	                    #sFB_Conveyor730(iUDT_ConveyorConfiguration := #iUDT_Configuration."730".Conveyor,
	                                     idi_PECEoSDistance := #iUDT_Configuration."730".PEC_Eos.Distance,
	                                     idi_PECBoSDistance := 0,
	                                     ii_ExternalSpeed := 0,
	                                     ix_SafetyOk := #ix_SafetyOk,
	                                     ix_24vOk := #ix_24vOk,
	                                     ix_400vOk := #ix_400vOk,
	                                     ix_HardwareOk := #ix_HardwareOk,
	                                     ix_PECEoS := #iqUDT_WorkstationStatus."730".PEC_EoS.PEC,
	                                     ix_PECBoS := TRUE,
	                                     ix_ReverseDirection := FALSE,
	                                     ix_ExternalRequestDieBack := FALSE,
	                                     ix_ExternalRequestHold := #sx_RightExternalRequestHold730,
	                                     ix_ResetEnergySave := FALSE,
	                                     qUDT_HMIStatus => #iqUDT_WorkstationStatus."730".Conveyor,
	                                     qUDT_Status => #iqUDT_WorkstationCommonStatus."730",
	                                     iqUDT_EquipmentControl := #iqUDT_EquipmentControl,
	                                     iqUDT_ConveyorCommand := #iqUDT_WorkstationCommands."730".Conveyor,
	                                     iqUDT_ConveyorInterface := #sUDT_Interface730,
	                                     iqUDT_HandShakeUp := #sUDT_Handshake720,
	                                     iqUDT_HandShake := #sUDT_Handshake730,
	                                     iqUDT_Statistics := #iqUDT_WorkstationStatistics."730".Conveyor);
	                END_REGION

	                REGION MCO

	                    #sFB_MCOConveyLinxAixController730(iUDT_AixConfig := #iUDT_Configuration."730".MCO_M01,
	                                                       iUDT_AixInputsModule := #iUDT_MotorInput730,
	                                                       ix_24vOk := #ix_24vOk,
	                                                       ix_SimulationModeActive := "DB_Memory".Simulation,
	                                                       ii_MotorPositionId := 1,
	                                                       qUDT_HMIStatus => #iqUDT_WorkstationStatus."730".MCO_M01,
	                                                       iqUDT_AixOutputsModule := #iqUDT_MotorOutput730,
	                                                       iqUDT_ConveyorInterface := #sUDT_Interface730,
	                                                       iqUDT_MCOStatistics := #iqUDT_WorkstationStatistics."730".MCO_M01);
	                END_REGION
	            END_REGION

	            REGION 740

	                REGION Displacement

	                    #sFB_Displacement740(#sUDT_Interface740);

	                END_REGION

	                REGION EOS
	                    #sFB_PEC740(ix_PEC := NOT #iUDT_MotorInput730.AllSensorPortInputs.RightSensor,
	                                iUDT_PECConfiguration := #iUDT_Configuration."740".PEC_Eos,
	                                qx_PECFiltered => #tx_dummy,
	                                qUDT_HMIStatus => #iqUDT_WorkstationStatus."740".PEC_EoS,
	                                iqUDT_ConveyorInterface := #sUDT_Interface740,
	                                iqUDT_PECStatistics := #iqUDT_WorkstationStatistics."740".PEC_EoS);


	                END_REGION


	                REGION Conveyor

	                    #sFB_Conveyor740(iUDT_ConveyorConfiguration := #iUDT_Configuration."740".Conveyor,
	                                     idi_PECEoSDistance := #iUDT_Configuration."740".PEC_Eos.Distance,
	                                     idi_PECBoSDistance := 0,
	                                     ii_ExternalSpeed := 0,
	                                     ix_SafetyOk := #ix_SafetyOk,
	                                     ix_24vOk := #ix_24vOk,
	                                     ix_400vOk := #ix_400vOk,
	                                     ix_HardwareOk := #ix_HardwareOk,
	                                     ix_PECEoS := #iqUDT_WorkstationStatus."740".PEC_EoS.PEC,
	                                     ix_PECBoS := TRUE,
	                                     ix_ReverseDirection := FALSE,
	                                     ix_ExternalRequestDieBack := FALSE,
	                                     ix_ExternalRequestHold := #sx_RightExternalRequestHold740,
	                                     ix_ResetEnergySave := FALSE,
	                                     qUDT_HMIStatus => #iqUDT_WorkstationStatus."740".Conveyor,
	                                     qUDT_Status => #iqUDT_WorkstationCommonStatus."740",
	                                     iqUDT_EquipmentControl := #iqUDT_EquipmentControl,
	                                     iqUDT_ConveyorCommand := #iqUDT_WorkstationCommands."740".Conveyor,
	                                     iqUDT_ConveyorInterface := #sUDT_Interface740,
	                                     iqUDT_HandShakeUp := #sUDT_Handshake730,
	                                     iqUDT_HandShake := #sUDT_Handshake740,
	                                     iqUDT_Statistics := #iqUDT_WorkstationStatistics."740".Conveyor);
	                END_REGION

	                REGION MCO

	                    #sFB_MCOConveyLinxAixController740(iUDT_AixConfig := #iUDT_Configuration."740".MCO_M01,
	                                                       iUDT_AixInputsModule := #iUDT_MotorInput730,
	                                                       ix_24vOk := #ix_24vOk,
	                                                       ix_SimulationModeActive := "DB_Memory".Simulation,
	                                                       ii_MotorPositionId := 2,
	                                                       qUDT_HMIStatus => #iqUDT_WorkstationStatus."740".MCO_M01,
	                                                       iqUDT_AixOutputsModule := #iqUDT_MotorOutput730,
	                                                       iqUDT_ConveyorInterface := #sUDT_Interface740,
	                                                       iqUDT_MCOStatistics := #iqUDT_WorkstationStatistics."740".MCO_M01);
	                END_REGION

	            END_REGION

	            REGION 750

	                REGION Displacement

	                    #sFB_Displacement750(#sUDT_Interface750);

	                END_REGION

	                REGION EOS
	                    #sFB_PEC750(ix_PEC := NOT #iUDT_MotorInput750.AllSensorPortInputs.LeftSensor,
	                                iUDT_PECConfiguration := #iUDT_Configuration."750".PEC_Eos,
	                                qx_PECFiltered => #tx_dummy,
	                                qUDT_HMIStatus => #iqUDT_WorkstationStatus."750".PEC_EoS,
	                                iqUDT_ConveyorInterface := #sUDT_Interface750,
	                                iqUDT_PECStatistics := #iqUDT_WorkstationStatistics."750".PEC_EoS);

	                END_REGION

	                REGION Conveyor

	                    #sUDT_Handshake750.RTR := #sUDT_Handshake750.RTR OR #iqUDT_WorkstationStatus."750".PEC_EoS.PEC;

	                    #sFB_Conveyor750(iUDT_ConveyorConfiguration := #iUDT_Configuration."750".Conveyor,
	                                     idi_PECEoSDistance := #iUDT_Configuration."750".PEC_Eos.Distance,
	                                     idi_PECBoSDistance := 0,
	                                     ii_ExternalSpeed := 0,
	                                     ix_SafetyOk := #ix_SafetyOk,
	                                     ix_24vOk := #ix_24vOk,
	                                     ix_400vOk := #ix_400vOk,
	                                     ix_HardwareOk := #ix_HardwareOk,
	                                     ix_PECEoS := #iqUDT_WorkstationStatus."750".PEC_EoS.PEC,
	                                     ix_PECBoS := TRUE,
	                                     ix_ReverseDirection := FALSE,
	                                     ix_ExternalRequestDieBack := FALSE,
	                                     ix_ExternalRequestHold := #sx_RightExternalRequestHold750,
	                                     ix_ResetEnergySave := FALSE,
	                                     qUDT_HMIStatus => #iqUDT_WorkstationStatus."750".Conveyor,
	                                     qUDT_Status => #iqUDT_WorkstationCommonStatus."750",
	                                     iqUDT_EquipmentControl := #iqUDT_EquipmentControl,
	                                     iqUDT_ConveyorCommand := #iqUDT_WorkstationCommands."750".Conveyor,
	                                     iqUDT_ConveyorInterface := #sUDT_Interface750,
	                                     iqUDT_HandShakeUp := #sUDT_Handshake740,
	                                     iqUDT_HandShake := #sUDT_Handshake750,
	                                     iqUDT_Statistics := #iqUDT_WorkstationStatistics."750".Conveyor);
	                END_REGION

	                REGION MCO

	                    #sFB_MCOConveyLinxAixController750(iUDT_AixConfig := #iUDT_Configuration."750".MCO_M01,
	                                                       iUDT_AixInputsModule := #iUDT_MotorInput750,
	                                                       ix_24vOk := #ix_24vOk,
	                                                       ix_SimulationModeActive := "DB_Memory".Simulation,
	                                                       ii_MotorPositionId := 1,
	                                                       qUDT_HMIStatus => #iqUDT_WorkstationStatus."750".MCO_M01,
	                                                       iqUDT_AixOutputsModule := #iqUDT_MotorOutput750,
	                                                       iqUDT_ConveyorInterface := #sUDT_Interface750,
	                                                       iqUDT_MCOStatistics := #iqUDT_WorkstationStatistics."750".MCO_M01);
	                END_REGION
	            END_REGION
	        END_REGION

	    END_IF;
	END_REGION

END_FUNCTION_BLOCK

FUNCTION_BLOCK "FB_WSR"
{ S7_Optimized_Access := 'TRUE' }
VERSION : 0.1
// ATTRIBUTES
// AUTO_NUMBER = True
// BLOCK_NUMBER = 270
// END_ATTRIBUTES
   VAR_INPUT
      iUDT_MotorInput010 { ExternalAccessible := 'False'; ExternalVisible := 'False'; ExternalWritable := 'False'} : "UDT_AixPlcFullIn";   // 010 ConveyLinxAix inputs structure
      iUDT_MotorInput030 { ExternalAccessible := 'False'; ExternalVisible := 'False'; ExternalWritable := 'False'} : "UDT_AixPlcFullIn";   // 030 ConveyLinxAix inputs structure
      iUDT_MotorInput040 { ExternalAccessible := 'False'; ExternalVisible := 'False'; ExternalWritable := 'False'} : "UDT_AixPlcFullIn";   // 040 ConveyLinxAix inputs structure
      iUDT_MotorInput050 { ExternalAccessible := 'False'; ExternalVisible := 'False'; ExternalWritable := 'False'} : "UDT_AixPlcFullIn";   // 050 ConveyLinxAix inputs structure
      iUDT_MotorInput070 { ExternalAccessible := 'False'; ExternalVisible := 'False'; ExternalWritable := 'False'} : "UDT_AixPlcFullIn";   // 070 ConveyLinxAix inputs structure
      iUDT_MotorInput110 { ExternalAccessible := 'False'; ExternalVisible := 'False'; ExternalWritable := 'False'} : "UDT_AixPlcFullIn";   // 110 ConveyLinxAix inputs structure
      iUDT_MotorInput130 { ExternalAccessible := 'False'; ExternalVisible := 'False'; ExternalWritable := 'False'} : "UDT_AixPlcFullIn";   // 130 ConveyLinxAix inputs structure
      iUDT_MotorInput140 { ExternalAccessible := 'False'; ExternalVisible := 'False'; ExternalWritable := 'False'} : "UDT_AixPlcFullIn";   // 140 ConveyLinxAix inputs structure
      iUDT_MotorInput150 { ExternalAccessible := 'False'; ExternalVisible := 'False'; ExternalWritable := 'False'} : "UDT_AixPlcFullIn";   // 150 ConveyLinxAix inputs structure
      iUDT_MotorInput170 { ExternalAccessible := 'False'; ExternalVisible := 'False'; ExternalWritable := 'False'} : "UDT_AixPlcFullIn";   // 170 ConveyLinxAix inputs structure
      iUDT_MotorInput210 { ExternalAccessible := 'False'; ExternalVisible := 'False'; ExternalWritable := 'False'} : "UDT_AixPlcFullIn";   // 210 ConveyLinxAix inputs structure
      iUDT_MotorInput230 { ExternalAccessible := 'False'; ExternalVisible := 'False'; ExternalWritable := 'False'} : "UDT_AixPlcFullIn";   // 230 ConveyLinxAix inputs structure
      iUDT_MotorInput240 { ExternalAccessible := 'False'; ExternalVisible := 'False'; ExternalWritable := 'False'} : "UDT_AixPlcFullIn";   // 240 ConveyLinxAix inputs structure
      iUDT_MotorInput250 { ExternalAccessible := 'False'; ExternalVisible := 'False'; ExternalWritable := 'False'} : "UDT_AixPlcFullIn";   // 250 ConveyLinxAix inputs structure
      iUDT_MotorInput270 { ExternalAccessible := 'False'; ExternalVisible := 'False'; ExternalWritable := 'False'} : "UDT_AixPlcFullIn";   // 270 ConveyLinxAix inputs structure
      ix_24vOk { ExternalAccessible := 'False'; ExternalVisible := 'False'; ExternalWritable := 'False'} : Bool;   // TRUE when 24VDC is healthy
      ix_400vOk { ExternalAccessible := 'False'; ExternalVisible := 'False'; ExternalWritable := 'False'} : Bool;   // TRUE when 400VAC is healthy
      ix_SafetyOk { ExternalAccessible := 'False'; ExternalVisible := 'False'; ExternalWritable := 'False'} : Bool;   // TRUE when safety is ok
      ix_HardwareOk { ExternalAccessible := 'False'; ExternalVisible := 'False'; ExternalWritable := 'False'} : Bool;   // TRUE when  hardware is ok
      ix_AirPressureOk { ExternalAccessible := 'False'; ExternalVisible := 'False'; ExternalWritable := 'False'} : Bool;   // TRUE when air pressure is ok
      ix_SectionisUp041 { ExternalAccessible := 'False'; ExternalVisible := 'False'; ExternalWritable := 'False'} : Bool;   // TRUE when 041 section is up
      ix_SectionisDown041 { ExternalAccessible := 'False'; ExternalVisible := 'False'; ExternalWritable := 'False'} : Bool;   // TRUE when 041 section is down
      ix_SectionisUp141 { ExternalAccessible := 'False'; ExternalVisible := 'False'; ExternalWritable := 'False'} : Bool;   // TRUE when 141 section is up
      ix_SectionisDown141 { ExternalAccessible := 'False'; ExternalVisible := 'False'; ExternalWritable := 'False'} : Bool;   // TRUE when 141 section is down
      ix_SectionisUp241 { ExternalAccessible := 'False'; ExternalVisible := 'False'; ExternalWritable := 'False'} : Bool;   // TRUE when 241 section is up
      ix_SectionisDown241 { ExternalAccessible := 'False'; ExternalVisible := 'False'; ExternalWritable := 'False'} : Bool;   // TRUE when 041 section is down
      ix_BladeStopisUp040 { ExternalAccessible := 'False'; ExternalVisible := 'False'; ExternalWritable := 'False'} : Bool;   // TRUE when 040 blade stop is up
      ix_BladeStopisDown040 { ExternalAccessible := 'False'; ExternalVisible := 'False'; ExternalWritable := 'False'} : Bool;   // TRUE when 040 blade stop is down
      ix_BladeStopisUp140 { ExternalAccessible := 'False'; ExternalVisible := 'False'; ExternalWritable := 'False'} : Bool;   // TRUE when 140 blade stop is up
      ix_BladeStopisDown140 { ExternalAccessible := 'False'; ExternalVisible := 'False'; ExternalWritable := 'False'} : Bool;   // TRUE when 140 blade stop is down
      ix_StationActive { ExternalAccessible := 'False'; ExternalVisible := 'False'; ExternalWritable := 'False'} : Bool;
   END_VAR

   VAR_OUTPUT
      qx_PopupControl041 { ExternalAccessible := 'False'; ExternalVisible := 'False'; ExternalWritable := 'False'} : Bool;   // Command up for section 041
      qx_PopupControl141 { ExternalAccessible := 'False'; ExternalVisible := 'False'; ExternalWritable := 'False'} : Bool;   // Command up for section 141
      qx_PopupControl241 { ExternalAccessible := 'False'; ExternalVisible := 'False'; ExternalWritable := 'False'} : Bool;   // Command up for section 241
      qx_BladeStopControl040 { ExternalAccessible := 'False'; ExternalVisible := 'False'; ExternalWritable := 'False'} : Bool;   // Command up for blade stop 040
      qx_BladeStopControl140 { ExternalAccessible := 'False'; ExternalVisible := 'False'; ExternalWritable := 'False'} : Bool;   // Command up for blade stop 140
   END_VAR

   VAR_IN_OUT
      iqUDT_Configuration : "UDT_WSRConfiguration";   // Workstation configuration structure
      iqUDT_EquipmentControl : "UDT_EquipmentControl";   // Equipment control structure
      iqUDT_HandshakeUpstream010 : "UDT_ConveyorHandshake";   // Upstream handshake structure in forward direction for 010 conveyor
      iqUDT_HandshakeUpstream110 : "UDT_ConveyorHandshake";   // Upstream handshake structure in forward direction for 110 conveyor
      iqUDT_HandshakeDownstream270 : "UDT_ConveyorHandshake";   // Handshake structure in forward direction for 270 conveyor
      iqUDT_UnknownGINRange : "UDT_UnknownGIN";   // Unknown GIN
      iqUDT_WorkstationCommands : "UDT_WSRHmiCommands";   // Workstation command structure
      iqUDT_WorkstationStatistics : "UDT_WSRStatistics";   // Statistics structure
      iqUDT_WorkstationStatus : "UDT_WSRStatus";   // HMI Status structure
      iqUDT_WorkstationCommonStatus : "UDT_WSRCommonStatus";   // Common status structure
      iqa_EmptyFifoHeader : "UDT_FifoHeader";
      iqa_EmptyFifoData : Array[*] of Int;
      iqa_PartialFifoHeader : "UDT_FifoHeader";
      iqa_PartialFifoData : Array[*] of Int;
      iqUDT_EmptyBuffer : "UDT_WSRBufferState";
      iqUDT_PartialBuffer : "UDT_WSRBufferState";
      iqi_Request030 { ExternalAccessible := 'False'; ExternalVisible := 'False'; ExternalWritable := 'False'} : Int;   // Request empty - 1 Request partialy - 2
      iqi_Request130 { ExternalAccessible := 'False'; ExternalVisible := 'False'; ExternalWritable := 'False'} : Int;   // Request empty - 1 Request partialy - 2
      iqx_ReleaseBin050 { ExternalAccessible := 'False'; ExternalVisible := 'False'; ExternalWritable := 'False'} : Bool;
      iqx_ReleaseBin060 { ExternalAccessible := 'False'; ExternalVisible := 'False'; ExternalWritable := 'False'} : Bool;
      iqx_ReleaseBin070 { ExternalAccessible := 'False'; ExternalVisible := 'False'; ExternalWritable := 'False'} : Bool;
      iqx_ReleaseBin150 { ExternalAccessible := 'False'; ExternalVisible := 'False'; ExternalWritable := 'False'} : Bool;
      iqx_ReleaseBin160 { ExternalAccessible := 'False'; ExternalVisible := 'False'; ExternalWritable := 'False'} : Bool;
      iqx_ReleaseBin170 { ExternalAccessible := 'False'; ExternalVisible := 'False'; ExternalWritable := 'False'} : Bool;
      iqUDT_MotorOutput010 : "UDT_AixPlcFullOut";   // 010 ConveyLinxAix outputs structure
      iqUDT_MotorOutput030 : "UDT_AixPlcFullOut";   // 030 ConveyLinxAix outputs structure
      iqUDT_MotorOutput040 : "UDT_AixPlcFullOut";   // 040 ConveyLinxAix outputs structure
      iqUDT_MotorOutput050 : "UDT_AixPlcFullOut";   // 050 ConveyLinxAix outputs structure
      iqUDT_MotorOutput070 : "UDT_AixPlcFullOut";   // 070 ConveyLinxAix outputs structure
      iqUDT_MotorOutput110 : "UDT_AixPlcFullOut";   // 110 ConveyLinxAix outputs structure
      iqUDT_MotorOutput130 : "UDT_AixPlcFullOut";   // 130 ConveyLinxAix outputs structure
      iqUDT_MotorOutput140 : "UDT_AixPlcFullOut";   // 140 ConveyLinxAix outputs structure
      iqUDT_MotorOutput150 : "UDT_AixPlcFullOut";   // 150 ConveyLinxAix outputs structure
      iqUDT_MotorOutput170 : "UDT_AixPlcFullOut";   // 170 ConveyLinxAix outputs structure
      iqUDT_MotorOutput210 : "UDT_AixPlcFullOut";   // 210 ConveyLinxAix outputs structure
      iqUDT_MotorOutput230 : "UDT_AixPlcFullOut";   // 230 ConveyLinxAix outputs structure
      iqUDT_MotorOutput240 : "UDT_AixPlcFullOut";   // 240 ConveyLinxAix outputs structure
      iqUDT_MotorOutput250 : "UDT_AixPlcFullOut";   // 250 ConveyLinxAix outputs structure
      iqUDT_MotorOutput270 : "UDT_AixPlcFullOut";   // 270 ConveyLinxAix outputs structure
      iqUDT_RATPositioning040 : "UDT_RATPositioning";   // Structure including data for servo control RAT 041
      iqUDT_RATPositioning140 : "UDT_RATPositioning";   // Structure including data for servo control RAT 141
      iqUDT_RATPositioning240 : "UDT_RATPositioning";   // Structure including data for servo control RAT 241
   END_VAR

   VAR
      sFB_Displacement010 { ExternalAccessible := 'False'; ExternalVisible := 'False'; ExternalWritable := 'False'; S7_SetPoint := 'False'} : "FB_Displacement";   // Displacement calculation for 010 conveyor
      sFB_Displacement020 { ExternalAccessible := 'False'; ExternalVisible := 'False'; ExternalWritable := 'False'; S7_SetPoint := 'False'} : "FB_Displacement";   // Displacement calculation for 020 conveyor
      sFB_Displacement030 { ExternalAccessible := 'False'; ExternalVisible := 'False'; ExternalWritable := 'False'; S7_SetPoint := 'False'} : "FB_Displacement";   // Displacement calculation for 030 conveyor
      sFB_Displacement040 { ExternalAccessible := 'False'; ExternalVisible := 'False'; ExternalWritable := 'False'; S7_SetPoint := 'False'} : "FB_Displacement";   // Displacement calculation for 040 conveyor
      sFB_Displacement041 { ExternalAccessible := 'False'; ExternalVisible := 'False'; ExternalWritable := 'False'; S7_SetPoint := 'False'} : "FB_Displacement";   // Displacement calculation for 041 conveyor
      sFB_Displacement050 { ExternalAccessible := 'False'; ExternalVisible := 'False'; ExternalWritable := 'False'; S7_SetPoint := 'False'} : "FB_Displacement";   // Displacement calculation for 050 conveyor
      sFB_Displacement060 { ExternalAccessible := 'False'; ExternalVisible := 'False'; ExternalWritable := 'False'; S7_SetPoint := 'False'} : "FB_Displacement";   // Displacement calculation for 060 conveyor
      sFB_Displacement070 { ExternalAccessible := 'False'; ExternalVisible := 'False'; ExternalWritable := 'False'; S7_SetPoint := 'False'} : "FB_Displacement";   // Displacement calculation for 070 conveyor
      sFB_Displacement080 { ExternalAccessible := 'False'; ExternalVisible := 'False'; ExternalWritable := 'False'; S7_SetPoint := 'False'} : "FB_Displacement";   // Displacement calculation for 080 conveyor
      sFB_Displacement110 { ExternalAccessible := 'False'; ExternalVisible := 'False'; ExternalWritable := 'False'; S7_SetPoint := 'False'} : "FB_Displacement";   // Displacement calculation for 110 conveyor
      sFB_Displacement120 { ExternalAccessible := 'False'; ExternalVisible := 'False'; ExternalWritable := 'False'; S7_SetPoint := 'False'} : "FB_Displacement";   // Displacement calculation for 120 conveyor
      sFB_Displacement130 { ExternalAccessible := 'False'; ExternalVisible := 'False'; ExternalWritable := 'False'; S7_SetPoint := 'False'} : "FB_Displacement";   // Displacement calculation for 130 conveyor
      sFB_Displacement140 { ExternalAccessible := 'False'; ExternalVisible := 'False'; ExternalWritable := 'False'; S7_SetPoint := 'False'} : "FB_Displacement";   // Displacement calculation for 140 conveyor
      sFB_Displacement141 { ExternalAccessible := 'False'; ExternalVisible := 'False'; ExternalWritable := 'False'; S7_SetPoint := 'False'} : "FB_Displacement";   // Displacement calculation for 141 conveyor
      sFB_Displacement150 { ExternalAccessible := 'False'; ExternalVisible := 'False'; ExternalWritable := 'False'; S7_SetPoint := 'False'} : "FB_Displacement";   // Displacement calculation for 150 conveyor
      sFB_Displacement160 { ExternalAccessible := 'False'; ExternalVisible := 'False'; ExternalWritable := 'False'; S7_SetPoint := 'False'} : "FB_Displacement";   // Displacement calculation for 160 conveyor
      sFB_Displacement170 { ExternalAccessible := 'False'; ExternalVisible := 'False'; ExternalWritable := 'False'; S7_SetPoint := 'False'} : "FB_Displacement";   // Displacement calculation for 170 conveyor
      sFB_Displacement180 { ExternalAccessible := 'False'; ExternalVisible := 'False'; ExternalWritable := 'False'; S7_SetPoint := 'False'} : "FB_Displacement";   // Displacement calculation for 180 conveyor
      sFB_Displacement210 { ExternalAccessible := 'False'; ExternalVisible := 'False'; ExternalWritable := 'False'; S7_SetPoint := 'False'} : "FB_Displacement";   // Displacement calculation for 210 conveyor
      sFB_Displacement220 { ExternalAccessible := 'False'; ExternalVisible := 'False'; ExternalWritable := 'False'; S7_SetPoint := 'False'} : "FB_Displacement";   // Displacement calculation for 220 conveyor
      sFB_Displacement230 { ExternalAccessible := 'False'; ExternalVisible := 'False'; ExternalWritable := 'False'; S7_SetPoint := 'False'} : "FB_Displacement";   // Displacement calculation for 230 conveyor
      sFB_Displacement240 { ExternalAccessible := 'False'; ExternalVisible := 'False'; ExternalWritable := 'False'; S7_SetPoint := 'False'} : "FB_Displacement";   // Displacement calculation for 240 conveyor
      sFB_Displacement241 { ExternalAccessible := 'False'; ExternalVisible := 'False'; ExternalWritable := 'False'; S7_SetPoint := 'False'} : "FB_Displacement";   // Displacement calculation for 241 conveyor
      sFB_Displacement250 { ExternalAccessible := 'False'; ExternalVisible := 'False'; ExternalWritable := 'False'; S7_SetPoint := 'False'} : "FB_Displacement";   // Displacement calculation for 250 conveyor
      sFB_Displacement260 { ExternalAccessible := 'False'; ExternalVisible := 'False'; ExternalWritable := 'False'; S7_SetPoint := 'False'} : "FB_Displacement";   // Displacement calculation for 260 conveyor
      sFB_Displacement270 { ExternalAccessible := 'False'; ExternalVisible := 'False'; ExternalWritable := 'False'; S7_SetPoint := 'False'} : "FB_Displacement";   // Displacement calculation for 270 conveyor
      sUDT_Interface_010 { ExternalAccessible := 'False'; ExternalVisible := 'False'; ExternalWritable := 'False'; S7_SetPoint := 'False'} : "UDT_ConveyorInterface";   // Interface structure for 010 conveyor
      sUDT_Interface_020 { ExternalAccessible := 'False'; ExternalVisible := 'False'; ExternalWritable := 'False'; S7_SetPoint := 'False'} : "UDT_ConveyorInterface";   // Interface structure for 020 conveyor
      sUDT_Interface_030 { ExternalAccessible := 'False'; ExternalVisible := 'False'; ExternalWritable := 'False'; S7_SetPoint := 'False'} : "UDT_ConveyorInterface";   // Interface structure for 030 conveyor
      sUDT_Interface_040 { ExternalAccessible := 'False'; ExternalVisible := 'False'; ExternalWritable := 'False'; S7_SetPoint := 'False'} : "UDT_ConveyorInterface";   // Interface structure for 040 conveyor
      sUDT_Interface_041 { ExternalAccessible := 'False'; ExternalVisible := 'False'; ExternalWritable := 'False'; S7_SetPoint := 'False'} : "UDT_ConveyorInterface";   // Interface structure for 041 conveyor
      sUDT_Interface_050 { ExternalAccessible := 'False'; ExternalVisible := 'False'; ExternalWritable := 'False'; S7_SetPoint := 'False'} : "UDT_ConveyorInterface";   // Interface structure for 050 conveyor
      sUDT_Interface_060 { ExternalAccessible := 'False'; ExternalVisible := 'False'; ExternalWritable := 'False'; S7_SetPoint := 'False'} : "UDT_ConveyorInterface";   // Interface structure for 060 conveyor
      sUDT_Interface_070 { ExternalAccessible := 'False'; ExternalVisible := 'False'; ExternalWritable := 'False'; S7_SetPoint := 'False'} : "UDT_ConveyorInterface";   // Interface structure for 070 conveyor
      sUDT_Interface_080 { ExternalAccessible := 'False'; ExternalVisible := 'False'; ExternalWritable := 'False'; S7_SetPoint := 'False'} : "UDT_ConveyorInterface";   // Interface structure for 080 conveyor
      sUDT_Interface_110 { ExternalAccessible := 'False'; ExternalVisible := 'False'; ExternalWritable := 'False'; S7_SetPoint := 'False'} : "UDT_ConveyorInterface";   // Interface structure for 110 conveyor
      sUDT_Interface_120 { ExternalAccessible := 'False'; ExternalVisible := 'False'; ExternalWritable := 'False'; S7_SetPoint := 'False'} : "UDT_ConveyorInterface";   // Interface structure for 120 conveyor
      sUDT_Interface_130 { ExternalAccessible := 'False'; ExternalVisible := 'False'; ExternalWritable := 'False'; S7_SetPoint := 'False'} : "UDT_ConveyorInterface";   // Interface structure for 130 conveyor
      sUDT_Interface_140 { ExternalAccessible := 'False'; ExternalVisible := 'False'; ExternalWritable := 'False'; S7_SetPoint := 'False'} : "UDT_ConveyorInterface";   // Interface structure for 140 conveyor
      sUDT_Interface_141 { ExternalAccessible := 'False'; ExternalVisible := 'False'; ExternalWritable := 'False'; S7_SetPoint := 'False'} : "UDT_ConveyorInterface";   // Interface structure for 141 conveyor
      sUDT_Interface_150 { ExternalAccessible := 'False'; ExternalVisible := 'False'; ExternalWritable := 'False'; S7_SetPoint := 'False'} : "UDT_ConveyorInterface";   // Interface structure for 150 conveyor
      sUDT_Interface_160 { ExternalAccessible := 'False'; ExternalVisible := 'False'; ExternalWritable := 'False'; S7_SetPoint := 'False'} : "UDT_ConveyorInterface";   // Interface structure for 160 conveyor
      sUDT_Interface_170 { ExternalAccessible := 'False'; ExternalVisible := 'False'; ExternalWritable := 'False'; S7_SetPoint := 'False'} : "UDT_ConveyorInterface";   // Interface structure for 170 conveyor
      sUDT_Interface_180 { ExternalAccessible := 'False'; ExternalVisible := 'False'; ExternalWritable := 'False'; S7_SetPoint := 'False'} : "UDT_ConveyorInterface";   // Interface structure for 180 conveyor
      sUDT_Interface_210 { ExternalAccessible := 'False'; ExternalVisible := 'False'; ExternalWritable := 'False'; S7_SetPoint := 'False'} : "UDT_ConveyorInterface";   // Interface structure for 210 conveyor
      sUDT_Interface_220 { ExternalAccessible := 'False'; ExternalVisible := 'False'; ExternalWritable := 'False'; S7_SetPoint := 'False'} : "UDT_ConveyorInterface";   // Interface structure for 220 conveyor
      sUDT_Interface_230 { ExternalAccessible := 'False'; ExternalVisible := 'False'; ExternalWritable := 'False'; S7_SetPoint := 'False'} : "UDT_ConveyorInterface";   // Interface structure for 230 conveyor
      sUDT_Interface_240 { ExternalAccessible := 'False'; ExternalVisible := 'False'; ExternalWritable := 'False'; S7_SetPoint := 'False'} : "UDT_ConveyorInterface";   // Interface structure for 240 conveyor
      sUDT_Interface_241 { ExternalAccessible := 'False'; ExternalVisible := 'False'; ExternalWritable := 'False'; S7_SetPoint := 'False'} : "UDT_ConveyorInterface";   // Interface structure for 241 conveyor
      sUDT_Interface_250 { ExternalAccessible := 'False'; ExternalVisible := 'False'; ExternalWritable := 'False'; S7_SetPoint := 'False'} : "UDT_ConveyorInterface";   // Interface structure for 250 conveyor
      sUDT_Interface_260 { ExternalAccessible := 'False'; ExternalVisible := 'False'; ExternalWritable := 'False'; S7_SetPoint := 'False'} : "UDT_ConveyorInterface";   // Interface structure for 260 conveyor
      sUDT_Interface_270 { ExternalAccessible := 'False'; ExternalVisible := 'False'; ExternalWritable := 'False'; S7_SetPoint := 'False'} : "UDT_ConveyorInterface";   // Interface structure for 270 conveyor
      sUDT_Interface_040_BladeStopEoS { ExternalAccessible := 'False'; ExternalVisible := 'False'; ExternalWritable := 'False'; S7_SetPoint := 'False'} : "UDT_ValveInterface";   // Interface structure for 040 blade stop
      sUDT_Interface_140_BladeStopEoS { ExternalAccessible := 'False'; ExternalVisible := 'False'; ExternalWritable := 'False'; S7_SetPoint := 'False'} : "UDT_ValveInterface";   // Interface structure for 140 blade stop
      sFB_Tracking_010 { ExternalAccessible := 'False'; ExternalVisible := 'False'; ExternalWritable := 'False'; S7_SetPoint := 'False'} : "FB_Tracking";   // Tracking function for 010 conveyor
      sFB_Tracking_020 { ExternalAccessible := 'False'; ExternalVisible := 'False'; ExternalWritable := 'False'; S7_SetPoint := 'False'} : "FB_Tracking";   // Tracking function for 020 conveyor
      sFB_Tracking_030 { ExternalAccessible := 'False'; ExternalVisible := 'False'; ExternalWritable := 'False'; S7_SetPoint := 'False'} : "FB_Tracking";   // Tracking function for 030 conveyor
      sFB_Tracking_050 { ExternalAccessible := 'False'; ExternalVisible := 'False'; ExternalWritable := 'False'; S7_SetPoint := 'False'} : "FB_Tracking";   // Tracking function for 050 conveyor
      sFB_Tracking_060 { ExternalAccessible := 'False'; ExternalVisible := 'False'; ExternalWritable := 'False'; S7_SetPoint := 'False'} : "FB_Tracking";   // Tracking function for 060 conveyor
      sFB_Tracking_070 { ExternalAccessible := 'False'; ExternalVisible := 'False'; ExternalWritable := 'False'; S7_SetPoint := 'False'} : "FB_Tracking";   // Tracking function for 070 conveyor
      sFB_Tracking_110 { ExternalAccessible := 'False'; ExternalVisible := 'False'; ExternalWritable := 'False'; S7_SetPoint := 'False'} : "FB_Tracking";   // Tracking function for 110 conveyor
      sFB_Tracking_120 { ExternalAccessible := 'False'; ExternalVisible := 'False'; ExternalWritable := 'False'; S7_SetPoint := 'False'} : "FB_Tracking";   // Tracking function for 120 conveyor
      sFB_Tracking_130 { ExternalAccessible := 'False'; ExternalVisible := 'False'; ExternalWritable := 'False'; S7_SetPoint := 'False'} : "FB_Tracking";   // Tracking function for 130 conveyor
      sFB_Tracking_150 { ExternalAccessible := 'False'; ExternalVisible := 'False'; ExternalWritable := 'False'; S7_SetPoint := 'False'} : "FB_Tracking";   // Tracking function for 150 conveyor
      sFB_Tracking_160 { ExternalAccessible := 'False'; ExternalVisible := 'False'; ExternalWritable := 'False'; S7_SetPoint := 'False'} : "FB_Tracking";   // Tracking function for 160 conveyor
      sFB_Tracking_170 { ExternalAccessible := 'False'; ExternalVisible := 'False'; ExternalWritable := 'False'; S7_SetPoint := 'False'} : "FB_Tracking";   // Tracking function for 170 conveyor
      sFB_Tracking_210 { ExternalAccessible := 'False'; ExternalVisible := 'False'; ExternalWritable := 'False'; S7_SetPoint := 'False'} : "FB_Tracking";   // Tracking function for 210 conveyor
      sFB_Tracking_220 { ExternalAccessible := 'False'; ExternalVisible := 'False'; ExternalWritable := 'False'; S7_SetPoint := 'False'} : "FB_Tracking";   // Tracking function for 220 conveyor
      sFB_Tracking_230 { ExternalAccessible := 'False'; ExternalVisible := 'False'; ExternalWritable := 'False'; S7_SetPoint := 'False'} : "FB_Tracking";   // Tracking function for 230 conveyor
      sFB_Tracking_250 { ExternalAccessible := 'False'; ExternalVisible := 'False'; ExternalWritable := 'False'; S7_SetPoint := 'False'} : "FB_Tracking";   // Tracking function for 250 conveyor
      sFB_Tracking_260 { ExternalAccessible := 'False'; ExternalVisible := 'False'; ExternalWritable := 'False'; S7_SetPoint := 'False'} : "FB_Tracking";   // Tracking function for 260 conveyor
      sFB_Tracking_270 { ExternalAccessible := 'False'; ExternalVisible := 'False'; ExternalWritable := 'False'; S7_SetPoint := 'False'} : "FB_Tracking";   // Tracking function for 270 conveyor
      sa_TrackingArray_010 { ExternalAccessible := 'False'; ExternalVisible := 'False'; ExternalWritable := 'False'} : Array[0..100] of Int;   // Tracking array for 010 conveyor
      sa_TrackingArray_020 { ExternalAccessible := 'False'; ExternalVisible := 'False'; ExternalWritable := 'False'} : Array[0..100] of Int;   // Tracking array for 020 conveyor
      sa_TrackingArray_030 { ExternalAccessible := 'False'; ExternalVisible := 'False'; ExternalWritable := 'False'} : Array[0..100] of Int;   // Tracking array for 030 conveyor
      sa_TrackingArray_050 { ExternalAccessible := 'False'; ExternalVisible := 'False'; ExternalWritable := 'False'} : Array[0..100] of Int;   // Tracking array for 050 conveyor
      sa_TrackingArray_060 { ExternalAccessible := 'False'; ExternalVisible := 'False'; ExternalWritable := 'False'} : Array[0..100] of Int;   // Tracking array for 060 conveyor
      sa_TrackingArray_070 { ExternalAccessible := 'False'; ExternalVisible := 'False'; ExternalWritable := 'False'} : Array[0..100] of Int;   // Tracking array for 070 conveyor
      sa_TrackingArray_110 { ExternalAccessible := 'False'; ExternalVisible := 'False'; ExternalWritable := 'False'} : Array[0..100] of Int;   // Tracking array for 110 conveyor
      sa_TrackingArray_120 { ExternalAccessible := 'False'; ExternalVisible := 'False'; ExternalWritable := 'False'} : Array[0..100] of Int;   // Tracking array for 120 conveyor
      sa_TrackingArray_130 { ExternalAccessible := 'False'; ExternalVisible := 'False'; ExternalWritable := 'False'} : Array[0..100] of Int;   // Tracking array for 130 conveyor
      sa_TrackingArray_150 { ExternalAccessible := 'False'; ExternalVisible := 'False'; ExternalWritable := 'False'} : Array[0..100] of Int;   // Tracking array for 150 conveyor
      sa_TrackingArray_160 { ExternalAccessible := 'False'; ExternalVisible := 'False'; ExternalWritable := 'False'} : Array[0..100] of Int;   // Tracking array for 160 conveyor
      sa_TrackingArray_170 { ExternalAccessible := 'False'; ExternalVisible := 'False'; ExternalWritable := 'False'} : Array[0..100] of Int;   // Tracking array for 170 conveyor
      sa_TrackingArray_210 { ExternalAccessible := 'False'; ExternalVisible := 'False'; ExternalWritable := 'False'} : Array[0..100] of Int;   // Tracking array for 210 conveyor
      sa_TrackingArray_220 { ExternalAccessible := 'False'; ExternalVisible := 'False'; ExternalWritable := 'False'} : Array[0..100] of Int;   // Tracking array for 220 conveyor
      sa_TrackingArray_230 { ExternalAccessible := 'False'; ExternalVisible := 'False'; ExternalWritable := 'False'} : Array[0..100] of Int;   // Tracking array for 230 conveyor
      sa_TrackingArray_250 { ExternalAccessible := 'False'; ExternalVisible := 'False'; ExternalWritable := 'False'} : Array[0..100] of Int;   // Tracking array for 250 conveyor
      sa_TrackingArray_260 { ExternalAccessible := 'False'; ExternalVisible := 'False'; ExternalWritable := 'False'} : Array[0..100] of Int;   // Tracking array for 260 conveyor
      sa_TrackingArray_270 { ExternalAccessible := 'False'; ExternalVisible := 'False'; ExternalWritable := 'False'} : Array[0..100] of Int;   // Tracking array for 270 conveyor
      sUDT_Handshake_010 { ExternalAccessible := 'False'; ExternalVisible := 'False'; ExternalWritable := 'False'; S7_SetPoint := 'False'} : "UDT_ConveyorHandshake";   // Handshake structure for 010 conveyor
      sUDT_Handshake_020 { ExternalAccessible := 'False'; ExternalVisible := 'False'; ExternalWritable := 'False'; S7_SetPoint := 'False'} : "UDT_ConveyorHandshake";   // Handshake structure for 020 conveyor
      sUDT_Handshake_030 { ExternalAccessible := 'False'; ExternalVisible := 'False'; ExternalWritable := 'False'; S7_SetPoint := 'False'} : "UDT_ConveyorHandshake";   // Handshake structure for 030 conveyor
      sUDT_Handshake_040 { ExternalAccessible := 'False'; ExternalVisible := 'False'; ExternalWritable := 'False'; S7_SetPoint := 'False'} : "UDT_ConveyorHandshake";   // Handshake structure for 040 conveyor
      sUDT_Handshake_041 { ExternalAccessible := 'False'; ExternalVisible := 'False'; ExternalWritable := 'False'; S7_SetPoint := 'False'} : "UDT_ConveyorHandshake";   // Handshake structure for 041 conveyor
      sUDT_HandshakeUp_041 { ExternalAccessible := 'False'; ExternalVisible := 'False'; ExternalWritable := 'False'; S7_SetPoint := 'False'} : "UDT_ConveyorHandshake";   // Handshake structure for 041 conveyor
      sUDT_Handshake_050 { ExternalAccessible := 'False'; ExternalVisible := 'False'; ExternalWritable := 'False'; S7_SetPoint := 'False'} : "UDT_ConveyorHandshake";   // Handshake structure for 050 conveyor
      sUDT_Handshake_060 { ExternalAccessible := 'False'; ExternalVisible := 'False'; ExternalWritable := 'False'; S7_SetPoint := 'False'} : "UDT_ConveyorHandshake";   // Handshake structure for 060 conveyor
      sUDT_Handshake_070 { ExternalAccessible := 'False'; ExternalVisible := 'False'; ExternalWritable := 'False'; S7_SetPoint := 'False'} : "UDT_ConveyorHandshake";   // Handshake structure for 070 conveyor
      sUDT_Handshake_080 { ExternalAccessible := 'False'; ExternalVisible := 'False'; ExternalWritable := 'False'; S7_SetPoint := 'False'} : "UDT_ConveyorHandshake";   // Handshake structure for 080 conveyor
      sUDT_HandshakeUp_080 { ExternalAccessible := 'False'; ExternalVisible := 'False'; ExternalWritable := 'False'; S7_SetPoint := 'False'} : "UDT_ConveyorHandshake";   // Handshake structure for 080 conveyor
      sUDT_Handshake_110 { ExternalAccessible := 'False'; ExternalVisible := 'False'; ExternalWritable := 'False'; S7_SetPoint := 'False'} : "UDT_ConveyorHandshake";   // Handshake structure for 110 conveyor
      sUDT_Handshake_120 { ExternalAccessible := 'False'; ExternalVisible := 'False'; ExternalWritable := 'False'; S7_SetPoint := 'False'} : "UDT_ConveyorHandshake";   // Handshake structure for 120 conveyor
      sUDT_Handshake_130 { ExternalAccessible := 'False'; ExternalVisible := 'False'; ExternalWritable := 'False'; S7_SetPoint := 'False'} : "UDT_ConveyorHandshake";   // Handshake structure for 130 conveyor
      sUDT_Handshake_140 { ExternalAccessible := 'False'; ExternalVisible := 'False'; ExternalWritable := 'False'; S7_SetPoint := 'False'} : "UDT_ConveyorHandshake";   // Handshake structure for 140 conveyor
      sUDT_Handshake_141 { ExternalAccessible := 'False'; ExternalVisible := 'False'; ExternalWritable := 'False'; S7_SetPoint := 'False'} : "UDT_ConveyorHandshake";   // Handshake structure for 141 conveyor
      sUDT_Handshake_150 { ExternalAccessible := 'False'; ExternalVisible := 'False'; ExternalWritable := 'False'; S7_SetPoint := 'False'} : "UDT_ConveyorHandshake";   // Handshake structure for 150 conveyor
      sUDT_Handshake_160 { ExternalAccessible := 'False'; ExternalVisible := 'False'; ExternalWritable := 'False'; S7_SetPoint := 'False'} : "UDT_ConveyorHandshake";   // Handshake structure for 160 conveyor
      sUDT_Handshake_170 { ExternalAccessible := 'False'; ExternalVisible := 'False'; ExternalWritable := 'False'; S7_SetPoint := 'False'} : "UDT_ConveyorHandshake";   // Handshake structure for 170 conveyor
      sUDT_Handshake_180 { ExternalAccessible := 'False'; ExternalVisible := 'False'; ExternalWritable := 'False'; S7_SetPoint := 'False'} : "UDT_ConveyorHandshake";   // Handshake structure for 180 conveyor
      sUDT_HandshakeUp_180 { ExternalAccessible := 'False'; ExternalVisible := 'False'; ExternalWritable := 'False'; S7_SetPoint := 'False'} : "UDT_ConveyorHandshake";   // Handshake structure for 180 conveyor
      sUDT_HandshakeUp_210 { ExternalAccessible := 'False'; ExternalVisible := 'False'; ExternalWritable := 'False'; S7_SetPoint := 'False'} : "UDT_ConveyorHandshake";   // Handshake structure for 210 conveyor
      sUDT_Handshake_210 { ExternalAccessible := 'False'; ExternalVisible := 'False'; ExternalWritable := 'False'; S7_SetPoint := 'False'} : "UDT_ConveyorHandshake";   // Handshake structure for 210 conveyor
      sUDT_Handshake_220 { ExternalAccessible := 'False'; ExternalVisible := 'False'; ExternalWritable := 'False'; S7_SetPoint := 'False'} : "UDT_ConveyorHandshake";   // Handshake structure for 220 conveyor
      sUDT_Handshake_230 { ExternalAccessible := 'False'; ExternalVisible := 'False'; ExternalWritable := 'False'; S7_SetPoint := 'False'} : "UDT_ConveyorHandshake";   // Handshake structure for 230 conveyor
      sUDT_Handshake_240 { ExternalAccessible := 'False'; ExternalVisible := 'False'; ExternalWritable := 'False'; S7_SetPoint := 'False'} : "UDT_ConveyorHandshake";   // Handshake structure for 240 conveyor
      sUDT_Handshake_241 { ExternalAccessible := 'False'; ExternalVisible := 'False'; ExternalWritable := 'False'; S7_SetPoint := 'False'} : "UDT_ConveyorHandshake";   // Handshake structure for 241 conveyor
      sUDT_Handshake_250 { ExternalAccessible := 'False'; ExternalVisible := 'False'; ExternalWritable := 'False'; S7_SetPoint := 'False'} : "UDT_ConveyorHandshake";   // Handshake structure for 250 conveyor
      sUDT_Handshake_260 { ExternalAccessible := 'False'; ExternalVisible := 'False'; ExternalWritable := 'False'; S7_SetPoint := 'False'} : "UDT_ConveyorHandshake";   // Handshake structure for 260 conveyor
      sFB_PECUpdate_010 { ExternalAccessible := 'False'; ExternalVisible := 'False'; ExternalWritable := 'False'; S7_SetPoint := 'False'} : "FB_PECUpdate";   // Photoeye handling for 010 conveyor
      sFB_PECUpdate_020 { ExternalAccessible := 'False'; ExternalVisible := 'False'; ExternalWritable := 'False'; S7_SetPoint := 'False'} : "FB_PECUpdate";   // Photoeye handling for 020 conveyor
      sFB_PECUpdate_030 { ExternalAccessible := 'False'; ExternalVisible := 'False'; ExternalWritable := 'False'; S7_SetPoint := 'False'} : "FB_PECUpdate";   // Photoeye handling for 030 conveyor
      sFB_PECUpdate_050 { ExternalAccessible := 'False'; ExternalVisible := 'False'; ExternalWritable := 'False'; S7_SetPoint := 'False'} : "FB_PECUpdate";   // Photoeye handling for 050 conveyor
      sFB_PECUpdate_060 { ExternalAccessible := 'False'; ExternalVisible := 'False'; ExternalWritable := 'False'; S7_SetPoint := 'False'} : "FB_PECUpdate";   // Photoeye handling for 060 conveyor
      sFB_PECUpdate_070 { ExternalAccessible := 'False'; ExternalVisible := 'False'; ExternalWritable := 'False'; S7_SetPoint := 'False'} : "FB_PECUpdate";   // Photoeye handling for 070 conveyor
      sFB_PECUpdate_110 { ExternalAccessible := 'False'; ExternalVisible := 'False'; ExternalWritable := 'False'; S7_SetPoint := 'False'} : "FB_PECUpdate";   // Photoeye handling for 110 conveyor
      sFB_PECUpdate_120 { ExternalAccessible := 'False'; ExternalVisible := 'False'; ExternalWritable := 'False'; S7_SetPoint := 'False'} : "FB_PECUpdate";   // Photoeye handling for 120 conveyor
      sFB_PECUpdate_130 { ExternalAccessible := 'False'; ExternalVisible := 'False'; ExternalWritable := 'False'; S7_SetPoint := 'False'} : "FB_PECUpdate";   // Photoeye handling for 130 conveyor
      sFB_PECUpdate_150 { ExternalAccessible := 'False'; ExternalVisible := 'False'; ExternalWritable := 'False'; S7_SetPoint := 'False'} : "FB_PECUpdate";   // Photoeye handling for 150 conveyor
      sFB_PECUpdate_160 { ExternalAccessible := 'False'; ExternalVisible := 'False'; ExternalWritable := 'False'; S7_SetPoint := 'False'} : "FB_PECUpdate";   // Photoeye handling for 160 conveyor
      sFB_PECUpdate_170 { ExternalAccessible := 'False'; ExternalVisible := 'False'; ExternalWritable := 'False'; S7_SetPoint := 'False'} : "FB_PECUpdate";   // Photoeye handling for 170 conveyor
      sFB_PECUpdate_210 { ExternalAccessible := 'False'; ExternalVisible := 'False'; ExternalWritable := 'False'; S7_SetPoint := 'False'} : "FB_PECUpdate";   // Photoeye handling for 210 conveyor
      sFB_PECUpdate_220 { ExternalAccessible := 'False'; ExternalVisible := 'False'; ExternalWritable := 'False'; S7_SetPoint := 'False'} : "FB_PECUpdate";   // Photoeye handling for 220 conveyor
      sFB_PECUpdate_230 { ExternalAccessible := 'False'; ExternalVisible := 'False'; ExternalWritable := 'False'; S7_SetPoint := 'False'} : "FB_PECUpdate";   // Photoeye handling for 230 conveyor
      sFB_PECUpdate_250 { ExternalAccessible := 'False'; ExternalVisible := 'False'; ExternalWritable := 'False'; S7_SetPoint := 'False'} : "FB_PECUpdate";   // Photoeye handling for 250 conveyor
      sFB_PECUpdate_260 { ExternalAccessible := 'False'; ExternalVisible := 'False'; ExternalWritable := 'False'; S7_SetPoint := 'False'} : "FB_PECUpdate";   // Photoeye handling for 260 conveyor
      sFB_PECUpdate_270 { ExternalAccessible := 'False'; ExternalVisible := 'False'; ExternalWritable := 'False'; S7_SetPoint := 'False'} : "FB_PECUpdate";   // Photoeye handling for 270 conveyor
      sFB_Conveyor_010 { ExternalAccessible := 'False'; ExternalVisible := 'False'; ExternalWritable := 'False'; S7_SetPoint := 'False'} : "FB_Conveyor";   // Function block to control the 010 conveyor
      sFB_Conveyor_020 { ExternalAccessible := 'False'; ExternalVisible := 'False'; ExternalWritable := 'False'; S7_SetPoint := 'False'} : "FB_Conveyor";   // Function block to control the 020 conveyor
      sFB_Conveyor_030 { ExternalAccessible := 'False'; ExternalVisible := 'False'; ExternalWritable := 'False'; S7_SetPoint := 'False'} : "FB_Conveyor";   // Function block to control the 030 conveyor
      sFB_Conveyor_050 { ExternalAccessible := 'False'; ExternalVisible := 'False'; ExternalWritable := 'False'; S7_SetPoint := 'False'} : "FB_Conveyor";   // Function block to control the 050 conveyor
      sFB_Conveyor_060 { ExternalAccessible := 'False'; ExternalVisible := 'False'; ExternalWritable := 'False'; S7_SetPoint := 'False'} : "FB_Conveyor";   // Function block to control the 060 conveyor
      sFB_Conveyor_070 { ExternalAccessible := 'False'; ExternalVisible := 'False'; ExternalWritable := 'False'; S7_SetPoint := 'False'} : "FB_Conveyor";   // Function block to control the 070 conveyor
      sFB_Conveyor_080 { ExternalAccessible := 'False'; ExternalVisible := 'False'; ExternalWritable := 'False'; S7_SetPoint := 'False'} : "FB_Conveyor";   // Function block to control the 080 conveyor
      sFB_Conveyor_110 { ExternalAccessible := 'False'; ExternalVisible := 'False'; ExternalWritable := 'False'; S7_SetPoint := 'False'} : "FB_Conveyor";   // Function block to control the 110 conveyor
      sFB_Conveyor_120 { ExternalAccessible := 'False'; ExternalVisible := 'False'; ExternalWritable := 'False'; S7_SetPoint := 'False'} : "FB_Conveyor";   // Function block to control the 120 conveyor
      sFB_Conveyor_130 { ExternalAccessible := 'False'; ExternalVisible := 'False'; ExternalWritable := 'False'; S7_SetPoint := 'False'} : "FB_Conveyor";   // Function block to control the 130 conveyor
      sFB_Conveyor_150 { ExternalAccessible := 'False'; ExternalVisible := 'False'; ExternalWritable := 'False'; S7_SetPoint := 'False'} : "FB_Conveyor";   // Function block to control the 150 conveyor
      sFB_Conveyor_160 { ExternalAccessible := 'False'; ExternalVisible := 'False'; ExternalWritable := 'False'; S7_SetPoint := 'False'} : "FB_Conveyor";   // Function block to control the 160 conveyor
      sFB_Conveyor_170 { ExternalAccessible := 'False'; ExternalVisible := 'False'; ExternalWritable := 'False'; S7_SetPoint := 'False'} : "FB_Conveyor";   // Function block to control the 170 conveyor
      sFB_Conveyor_180 { ExternalAccessible := 'False'; ExternalVisible := 'False'; ExternalWritable := 'False'; S7_SetPoint := 'False'} : "FB_Conveyor";   // Function block to control the 180 conveyor
      sFB_Conveyor_210 { ExternalAccessible := 'False'; ExternalVisible := 'False'; ExternalWritable := 'False'; S7_SetPoint := 'False'} : "FB_Conveyor";   // Function block to control the 210 conveyor
      sFB_Conveyor_220 { ExternalAccessible := 'False'; ExternalVisible := 'False'; ExternalWritable := 'False'; S7_SetPoint := 'False'} : "FB_Conveyor";   // Function block to control the 220 conveyor
      sFB_Conveyor_230 { ExternalAccessible := 'False'; ExternalVisible := 'False'; ExternalWritable := 'False'; S7_SetPoint := 'False'} : "FB_Conveyor";   // Function block to control the 230 conveyor
      sFB_Conveyor_250 { ExternalAccessible := 'False'; ExternalVisible := 'False'; ExternalWritable := 'False'; S7_SetPoint := 'False'} : "FB_Conveyor";   // Function block to control the 250 conveyor
      sFB_Conveyor_260 { ExternalAccessible := 'False'; ExternalVisible := 'False'; ExternalWritable := 'False'; S7_SetPoint := 'False'} : "FB_Conveyor";   // Function block to control the 260 conveyor
      sFB_Conveyor_270 { ExternalAccessible := 'False'; ExternalVisible := 'False'; ExternalWritable := 'False'; S7_SetPoint := 'False'} : "FB_Conveyor";   // Function block to control the 270 conveyor
      sFB_MCOConveyLinxAixController_010 { ExternalAccessible := 'False'; ExternalVisible := 'False'; ExternalWritable := 'False'; S7_SetPoint := 'False'} : "FB_MCOConveyLinxAixController";   // Function to interface with ConveyLinx Aix Controller for 010
      sFB_MCOConveyLinxAixController_020 { ExternalAccessible := 'False'; ExternalVisible := 'False'; ExternalWritable := 'False'; S7_SetPoint := 'False'} : "FB_MCOConveyLinxAixController";   // Function to interface with ConveyLinx Aix Controller for 010
      sFB_MCOConveyLinxAixController_030 { ExternalAccessible := 'False'; ExternalVisible := 'False'; ExternalWritable := 'False'; S7_SetPoint := 'False'} : "FB_MCOConveyLinxAixController";   // Function to interface with ConveyLinx Aix Controller for 030
      sFB_MCOConveyLinxAixController_040 { ExternalAccessible := 'False'; ExternalVisible := 'False'; ExternalWritable := 'False'; S7_SetPoint := 'False'} : "FB_MCOConveyLinxAixController";   // Function to interface with ConveyLinx Aix Controller for 040
      sFB_MCOConveyLinxAixController_041 { ExternalAccessible := 'False'; ExternalVisible := 'False'; ExternalWritable := 'False'; S7_SetPoint := 'False'} : "FB_MCOConveyLinxAixController";   // Function to interface with ConveyLinx Aix Controller for 040
      sFB_MCOConveyLinxAixController_050 { ExternalAccessible := 'False'; ExternalVisible := 'False'; ExternalWritable := 'False'; S7_SetPoint := 'False'} : "FB_MCOConveyLinxAixController";   // Function to interface with ConveyLinx Aix Controller for 050
      sFB_MCOConveyLinxAixController_060 { ExternalAccessible := 'False'; ExternalVisible := 'False'; ExternalWritable := 'False'; S7_SetPoint := 'False'} : "FB_MCOConveyLinxAixController";   // Function to interface with ConveyLinx Aix Controller for 050
      sFB_MCOConveyLinxAixController_070 { ExternalAccessible := 'False'; ExternalVisible := 'False'; ExternalWritable := 'False'; S7_SetPoint := 'False'} : "FB_MCOConveyLinxAixController";   // Function to interface with ConveyLinx Aix Controller for 070
      sFB_MCOConveyLinxAixController_080 { ExternalAccessible := 'False'; ExternalVisible := 'False'; ExternalWritable := 'False'; S7_SetPoint := 'False'} : "FB_MCOConveyLinxAixController";   // Function to interface with ConveyLinx Aix Controller for 070
      sFB_MCOConveyLinxAixController_110 { ExternalAccessible := 'False'; ExternalVisible := 'False'; ExternalWritable := 'False'; S7_SetPoint := 'False'} : "FB_MCOConveyLinxAixController";   // Function to interface with ConveyLinx Aix Controller for 110
      sFB_MCOConveyLinxAixController_120 { ExternalAccessible := 'False'; ExternalVisible := 'False'; ExternalWritable := 'False'; S7_SetPoint := 'False'} : "FB_MCOConveyLinxAixController";   // Function to interface with ConveyLinx Aix Controller for 110
      sFB_MCOConveyLinxAixController_130 { ExternalAccessible := 'False'; ExternalVisible := 'False'; ExternalWritable := 'False'; S7_SetPoint := 'False'} : "FB_MCOConveyLinxAixController";   // Function to interface with ConveyLinx Aix Controller for 130
      sFB_MCOConveyLinxAixController_140 { ExternalAccessible := 'False'; ExternalVisible := 'False'; ExternalWritable := 'False'; S7_SetPoint := 'False'} : "FB_MCOConveyLinxAixController";   // Function to interface with ConveyLinx Aix Controller for 140
      sFB_MCOConveyLinxAixController_141 { ExternalAccessible := 'False'; ExternalVisible := 'False'; ExternalWritable := 'False'; S7_SetPoint := 'False'} : "FB_MCOConveyLinxAixController";   // Function to interface with ConveyLinx Aix Controller for 140
      sFB_MCOConveyLinxAixController_150 { ExternalAccessible := 'False'; ExternalVisible := 'False'; ExternalWritable := 'False'; S7_SetPoint := 'False'} : "FB_MCOConveyLinxAixController";   // Function to interface with ConveyLinx Aix Controller for 150
      sFB_MCOConveyLinxAixController_160 { ExternalAccessible := 'False'; ExternalVisible := 'False'; ExternalWritable := 'False'; S7_SetPoint := 'False'} : "FB_MCOConveyLinxAixController";   // Function to interface with ConveyLinx Aix Controller for 110
      sFB_MCOConveyLinxAixController_170 { ExternalAccessible := 'False'; ExternalVisible := 'False'; ExternalWritable := 'False'; S7_SetPoint := 'False'} : "FB_MCOConveyLinxAixController";   // Function to interface with ConveyLinx Aix Controller for 170
      sFB_MCOConveyLinxAixController_180 { ExternalAccessible := 'False'; ExternalVisible := 'False'; ExternalWritable := 'False'; S7_SetPoint := 'False'} : "FB_MCOConveyLinxAixController";   // Function to interface with ConveyLinx Aix Controller for 070
      sFB_MCOConveyLinxAixController_210 { ExternalAccessible := 'False'; ExternalVisible := 'False'; ExternalWritable := 'False'; S7_SetPoint := 'False'} : "FB_MCOConveyLinxAixController";   // Function to interface with ConveyLinx Aix Controller for 210
      sFB_MCOConveyLinxAixController_220 { ExternalAccessible := 'False'; ExternalVisible := 'False'; ExternalWritable := 'False'; S7_SetPoint := 'False'} : "FB_MCOConveyLinxAixController";   // Function to interface with ConveyLinx Aix Controller for 110
      sFB_MCOConveyLinxAixController_230 { ExternalAccessible := 'False'; ExternalVisible := 'False'; ExternalWritable := 'False'; S7_SetPoint := 'False'} : "FB_MCOConveyLinxAixController";   // Function to interface with ConveyLinx Aix Controller for 230
      sFB_MCOConveyLinxAixController_240 { ExternalAccessible := 'False'; ExternalVisible := 'False'; ExternalWritable := 'False'; S7_SetPoint := 'False'} : "FB_MCOConveyLinxAixController";   // Function to interface with ConveyLinx Aix Controller for 240
      sFB_MCOConveyLinxAixController_241 { ExternalAccessible := 'False'; ExternalVisible := 'False'; ExternalWritable := 'False'; S7_SetPoint := 'False'} : "FB_MCOConveyLinxAixController";   // Function to interface with ConveyLinx Aix Controller for 240
      sFB_MCOConveyLinxAixController_250 { ExternalAccessible := 'False'; ExternalVisible := 'False'; ExternalWritable := 'False'; S7_SetPoint := 'False'} : "FB_MCOConveyLinxAixController";   // Function to interface with ConveyLinx Aix Controller for 250
      sFB_MCOConveyLinxAixController_260 { ExternalAccessible := 'False'; ExternalVisible := 'False'; ExternalWritable := 'False'; S7_SetPoint := 'False'} : "FB_MCOConveyLinxAixController";   // Function to interface with ConveyLinx Aix Controller for 110
      sFB_MCOConveyLinxAixController_270 { ExternalAccessible := 'False'; ExternalVisible := 'False'; ExternalWritable := 'False'; S7_SetPoint := 'False'} : "FB_MCOConveyLinxAixController";   // Function to interface with ConveyLinx Aix Controller for 270
      sFB_BladeStopEoS_040 { ExternalAccessible := 'False'; ExternalVisible := 'False'; ExternalWritable := 'False'; S7_SetPoint := 'False'} : "FB_Valve";   // Function block to control the 040 blade stop
      sFB_BladeStopEoS_140 { ExternalAccessible := 'False'; ExternalVisible := 'False'; ExternalWritable := 'False'; S7_SetPoint := 'False'} : "FB_Valve";   // Function block to control the 140 blade stop
      sFB_RightAngledTransfer_041 { ExternalAccessible := 'False'; ExternalVisible := 'False'; ExternalWritable := 'False'; S7_SetPoint := 'False'} : "FB_RightAngledTransfer";   // Funtion to control 041 RAT
      sFB_RightAngledTransfer_141 { ExternalAccessible := 'False'; ExternalVisible := 'False'; ExternalWritable := 'False'; S7_SetPoint := 'False'} : "FB_RightAngledTransfer";   // Funtion to control 141 RAT
      sFB_RightAngledTransfer_241 { ExternalAccessible := 'False'; ExternalVisible := 'False'; ExternalWritable := 'False'; S7_SetPoint := 'False'} : "FB_RightAngledTransfer";   // Funtion to control 241 RAT
      sFB_OperationTimeout { ExternalAccessible := 'False'; ExternalVisible := 'False'; ExternalWritable := 'False'; S7_SetPoint := 'False'} : "FB_TimerOnOffDelay";   // Function block to generate operation timeout
      sF_TRIG_ParcelArrived1X0 {InstructionName := 'F_TRIG'; LibVersion := '1.0'; ExternalAccessible := 'False'; ExternalVisible := 'False'; ExternalWritable := 'False'; S7_SetPoint := 'False'} : F_TRIG;   // Parcel arrived on target detection 150
      sF_TRIG_ParcelArrived0X0 {InstructionName := 'F_TRIG'; LibVersion := '1.0'; ExternalAccessible := 'False'; ExternalVisible := 'False'; ExternalWritable := 'False'; S7_SetPoint := 'False'} : F_TRIG;   // Parcel arrived on target detection 050
      sF_TRIG_ParcelArrived2X0 {InstructionName := 'F_TRIG'; LibVersion := '1.0'; ExternalAccessible := 'False'; ExternalVisible := 'False'; ExternalWritable := 'False'; S7_SetPoint := 'False'} : F_TRIG;   // Parcel arrived on target detection 250
      sR_TRIG_NewParcel010 {InstructionName := 'R_TRIG'; LibVersion := '1.0'; ExternalAccessible := 'False'; ExternalVisible := 'False'; ExternalWritable := 'False'} : R_TRIG;
      sR_TRIG_NewParcel110 {InstructionName := 'R_TRIG'; LibVersion := '1.0'; ExternalAccessible := 'False'; ExternalVisible := 'False'; ExternalWritable := 'False'} : R_TRIG;
      si_EmptyBinRequiredCounter0X0 { ExternalAccessible := 'False'; ExternalVisible := 'False'; ExternalWritable := 'False'} : Int;   // Number of available empty bin request to 050 conveyor
      si_EmptyBinRequiredCounter1X0 { ExternalAccessible := 'False'; ExternalVisible := 'False'; ExternalWritable := 'False'} : Int;   // Number of available empty bin request to 150 conveyor
      si_PartialyBinRequiredCounter0X0 { ExternalAccessible := 'False'; ExternalVisible := 'False'; ExternalWritable := 'False'} : Int;   // Number of available partialy bin request to 050 conveyor
      si_PartialyBinRequiredCounter1X0 { ExternalAccessible := 'False'; ExternalVisible := 'False'; ExternalWritable := 'False'} : Int;   // Number of available partialy bin request to 050 conveyor
      si_040DestinationA { ExternalAccessible := 'False'; ExternalVisible := 'False'; ExternalWritable := 'False'} : Int;   // 040 RAT A destination value
      si_040DestinationB { ExternalAccessible := 'False'; ExternalVisible := 'False'; ExternalWritable := 'False'} : Int;   // 040 RAT B destination value
      si_040DestinationC { ExternalAccessible := 'False'; ExternalVisible := 'False'; ExternalWritable := 'False'} : Int;   // 040 RAT C destination value
      si_040DestinationD { ExternalAccessible := 'False'; ExternalVisible := 'False'; ExternalWritable := 'False'} : Int;   // 040 RAT D destination value
      si_140DestinationA { ExternalAccessible := 'False'; ExternalVisible := 'False'; ExternalWritable := 'False'} : Int;   // 140 RAT A destination value
      si_140DestinationB { ExternalAccessible := 'False'; ExternalVisible := 'False'; ExternalWritable := 'False'} : Int;   // 140 RAT B destination value
      si_140DestinationC { ExternalAccessible := 'False'; ExternalVisible := 'False'; ExternalWritable := 'False'} : Int;   // 140 RAT C destination value
      si_140DestinationD { ExternalAccessible := 'False'; ExternalVisible := 'False'; ExternalWritable := 'False'} : Int;   // 140 RAT D destination value
      si_240DestinationA { ExternalAccessible := 'False'; ExternalVisible := 'False'; ExternalWritable := 'False'} : Int;   // 240 RAT A destination value
      si_240DestinationB { ExternalAccessible := 'False'; ExternalVisible := 'False'; ExternalWritable := 'False'} : Int;   // 240 RAT B destination value
      si_240DestinationC { ExternalAccessible := 'False'; ExternalVisible := 'False'; ExternalWritable := 'False'} : Int;   // 240 RAT C destination value
      si_240DestinationD { ExternalAccessible := 'False'; ExternalVisible := 'False'; ExternalWritable := 'False'} : Int;   // 240 RAT D destination value
      sx_NoOperationInProgress { ExternalAccessible := 'False'; ExternalVisible := 'False'; ExternalWritable := 'False'} : Bool;   // No transfer active
      sx_Enable0X0In { ExternalAccessible := 'False'; ExternalVisible := 'False'; ExternalWritable := 'False'} : Bool;   // Enable 030 infeed
      sx_Enable1X0In { ExternalAccessible := 'False'; ExternalVisible := 'False'; ExternalWritable := 'False'} : Bool;   // Enable 130 infeed
      sx_Enable2X0In { ExternalAccessible := 'False'; ExternalVisible := 'False'; ExternalWritable := 'False'} : Bool;   // Enable 230 infeed
      si_SendTo0X0 { ExternalAccessible := 'False'; ExternalVisible := 'False'; ExternalWritable := 'False'} : Bool;   // Send to 050 active
      si_SendTo1X0 { ExternalAccessible := 'False'; ExternalVisible := 'False'; ExternalWritable := 'False'} : Bool;   // Send to 150 active
      si_SendTo2X0 { ExternalAccessible := 'False'; ExternalVisible := 'False'; ExternalWritable := 'False'} : Bool;   // Send to 250 active
      sx_Hold130 { ExternalAccessible := 'False'; ExternalVisible := 'False'; ExternalWritable := 'False'} : Bool;   // Hold 130 conveyor active
      sx_Hold030 { ExternalAccessible := 'False'; ExternalVisible := 'False'; ExternalWritable := 'False'} : Bool;   // Hold 030 conveyor active
      sx_Hold020 { ExternalAccessible := 'False'; ExternalVisible := 'False'; ExternalWritable := 'False'} : Bool;   // Hold 020 conveyor active
      sx_Hold120 { ExternalAccessible := 'False'; ExternalVisible := 'False'; ExternalWritable := 'False'} : Bool;   // Hold 120 conveyor active
      sx_Hold230 { ExternalAccessible := 'False'; ExternalVisible := 'False'; ExternalWritable := 'False'} : Bool;   // Hold 230 conveyor active
      sx_Hold220 { ExternalAccessible := 'False'; ExternalVisible := 'False'; ExternalWritable := 'False'} : Bool;   // Hold 220 conveyor active
      si_ReqestNewEmptyBin { ExternalAccessible := 'False'; ExternalVisible := 'False'; ExternalWritable := 'False'} : Int;
      si_ReqestNewPartialBin { ExternalAccessible := 'False'; ExternalVisible := 'False'; ExternalWritable := 'False'} : Int;
      si_LastGIN010 { ExternalAccessible := 'False'; ExternalVisible := 'False'; ExternalWritable := 'False'} : Int;
      si_LastGIN110 { ExternalAccessible := 'False'; ExternalVisible := 'False'; ExternalWritable := 'False'} : Int;
      sR_TRIG_EmptyBinReceived {InstructionName := 'R_TRIG'; LibVersion := '1.0'; ExternalAccessible := 'False'; ExternalVisible := 'False'; ExternalWritable := 'False'; S7_SetPoint := 'False'} : R_TRIG;
      sR_TRIG_PartialBinReceived {InstructionName := 'R_TRIG'; LibVersion := '1.0'; ExternalAccessible := 'False'; ExternalVisible := 'False'; ExternalWritable := 'False'; S7_SetPoint := 'False'} : R_TRIG;
      sR_TRIG_PartialBinReceived_1 {InstructionName := 'R_TRIG'; LibVersion := '1.0'; ExternalAccessible := 'False'; ExternalVisible := 'False'; ExternalWritable := 'False'; S7_SetPoint := 'False'} : R_TRIG;
      sR_TRIG_PartialBinReceived_2 {InstructionName := 'R_TRIG'; LibVersion := '1.0'; ExternalAccessible := 'False'; ExternalVisible := 'False'; ExternalWritable := 'False'; S7_SetPoint := 'False'} : R_TRIG;
      sR_TRIG_PartialBinReceived_3 {InstructionName := 'R_TRIG'; LibVersion := '1.0'; ExternalAccessible := 'False'; ExternalVisible := 'False'; ExternalWritable := 'False'; S7_SetPoint := 'False'} : R_TRIG;
      sR_TRIG_PartialBinReceived_4 {InstructionName := 'R_TRIG'; LibVersion := '1.0'; ExternalAccessible := 'False'; ExternalVisible := 'False'; ExternalWritable := 'False'; S7_SetPoint := 'False'} : R_TRIG;
      sR_TRIG_PartialBinReceived_5 {InstructionName := 'R_TRIG'; LibVersion := '1.0'; ExternalAccessible := 'False'; ExternalVisible := 'False'; ExternalWritable := 'False'; S7_SetPoint := 'False'} : R_TRIG;
      sR_TRIG_PartialBinReceived_6 {InstructionName := 'R_TRIG'; LibVersion := '1.0'; ExternalAccessible := 'False'; ExternalVisible := 'False'; ExternalWritable := 'False'; S7_SetPoint := 'False'} : R_TRIG;
      sR_TRIG_PartialBinReceived_7 {InstructionName := 'R_TRIG'; LibVersion := '1.0'; ExternalAccessible := 'False'; ExternalVisible := 'False'; ExternalWritable := 'False'; S7_SetPoint := 'False'} : R_TRIG;
      sR_TRIG_PartialBinReceived_8 {InstructionName := 'R_TRIG'; LibVersion := '1.0'; ExternalAccessible := 'False'; ExternalVisible := 'False'; ExternalWritable := 'False'; S7_SetPoint := 'False'} : R_TRIG;
      sR_TRIG_PartialBinReceived_9 {InstructionName := 'R_TRIG'; LibVersion := '1.0'; ExternalAccessible := 'False'; ExternalVisible := 'False'; ExternalWritable := 'False'; S7_SetPoint := 'False'} : R_TRIG;
      sR_TRIG_PartialBinReceived_10 {InstructionName := 'R_TRIG'; LibVersion := '1.0'; ExternalAccessible := 'False'; ExternalVisible := 'False'; ExternalWritable := 'False'; S7_SetPoint := 'False'} : R_TRIG;
      sR_TRIG_PartialBinReceived_11 {InstructionName := 'R_TRIG'; LibVersion := '1.0'; ExternalAccessible := 'False'; ExternalVisible := 'False'; ExternalWritable := 'False'; S7_SetPoint := 'False'} : R_TRIG;
      sR_TRIG_PartialBinReceived_12 {InstructionName := 'R_TRIG'; LibVersion := '1.0'; ExternalAccessible := 'False'; ExternalVisible := 'False'; ExternalWritable := 'False'; S7_SetPoint := 'False'} : R_TRIG;
      sR_TRIG_PartialBinReceived_13 {InstructionName := 'R_TRIG'; LibVersion := '1.0'; ExternalAccessible := 'False'; ExternalVisible := 'False'; ExternalWritable := 'False'; S7_SetPoint := 'False'} : R_TRIG;
      sR_TRIG_PartialBinReceived_14 {InstructionName := 'R_TRIG'; LibVersion := '1.0'; ExternalAccessible := 'False'; ExternalVisible := 'False'; ExternalWritable := 'False'; S7_SetPoint := 'False'} : R_TRIG;
      sR_TRIG_PartialBinReceived_15 {InstructionName := 'R_TRIG'; LibVersion := '1.0'; ExternalAccessible := 'False'; ExternalVisible := 'False'; ExternalWritable := 'False'; S7_SetPoint := 'False'} : R_TRIG;
      sR_TRIG_PartialBinReceived_16 {InstructionName := 'R_TRIG'; LibVersion := '1.0'; ExternalAccessible := 'False'; ExternalVisible := 'False'; ExternalWritable := 'False'; S7_SetPoint := 'False'} : R_TRIG;
      sR_TRIG_PartialBinReceived_17 {InstructionName := 'R_TRIG'; LibVersion := '1.0'; ExternalAccessible := 'False'; ExternalVisible := 'False'; ExternalWritable := 'False'; S7_SetPoint := 'False'} : R_TRIG;
      sR_TRIG_PartialBinReceived_18 {InstructionName := 'R_TRIG'; LibVersion := '1.0'; ExternalAccessible := 'False'; ExternalVisible := 'False'; ExternalWritable := 'False'; S7_SetPoint := 'False'} : R_TRIG;
      sR_TRIG_PartialBinReceived_19 {InstructionName := 'R_TRIG'; LibVersion := '1.0'; ExternalAccessible := 'False'; ExternalVisible := 'False'; ExternalWritable := 'False'; S7_SetPoint := 'False'} : R_TRIG;
      sR_TRIG_PartialBinReceived_20 {InstructionName := 'R_TRIG'; LibVersion := '1.0'; ExternalAccessible := 'False'; ExternalVisible := 'False'; ExternalWritable := 'False'; S7_SetPoint := 'False'} : R_TRIG;
      sR_TRIG_PartialBinReceived_21 {InstructionName := 'R_TRIG'; LibVersion := '1.0'; ExternalAccessible := 'False'; ExternalVisible := 'False'; ExternalWritable := 'False'; S7_SetPoint := 'False'} : R_TRIG;
      sR_TRIG_PartialBinReceived_22 {InstructionName := 'R_TRIG'; LibVersion := '1.0'; ExternalAccessible := 'False'; ExternalVisible := 'False'; ExternalWritable := 'False'; S7_SetPoint := 'False'} : R_TRIG;
      sR_TRIG_PartialBinReceived_23 {InstructionName := 'R_TRIG'; LibVersion := '1.0'; ExternalAccessible := 'False'; ExternalVisible := 'False'; ExternalWritable := 'False'; S7_SetPoint := 'False'} : R_TRIG;
      sR_TRIG_PartialBinReceived_24 {InstructionName := 'R_TRIG'; LibVersion := '1.0'; ExternalAccessible := 'False'; ExternalVisible := 'False'; ExternalWritable := 'False'; S7_SetPoint := 'False'} : R_TRIG;
      sR_TRIG_PartialBinReceived_25 {InstructionName := 'R_TRIG'; LibVersion := '1.0'; ExternalAccessible := 'False'; ExternalVisible := 'False'; ExternalWritable := 'False'; S7_SetPoint := 'False'} : R_TRIG;
      sR_TRIG_PartialBinReceived_26 {InstructionName := 'R_TRIG'; LibVersion := '1.0'; ExternalAccessible := 'False'; ExternalVisible := 'False'; ExternalWritable := 'False'; S7_SetPoint := 'False'} : R_TRIG;
      sR_TRIG_PartialBinReceived_27 {InstructionName := 'R_TRIG'; LibVersion := '1.0'; ExternalAccessible := 'False'; ExternalVisible := 'False'; ExternalWritable := 'False'; S7_SetPoint := 'False'} : R_TRIG;
      sR_TRIG_PartialBinReceived_28 {InstructionName := 'R_TRIG'; LibVersion := '1.0'; ExternalAccessible := 'False'; ExternalVisible := 'False'; ExternalWritable := 'False'; S7_SetPoint := 'False'} : R_TRIG;
      sR_TRIG_PartialBinReceived_29 {InstructionName := 'R_TRIG'; LibVersion := '1.0'; ExternalAccessible := 'False'; ExternalVisible := 'False'; ExternalWritable := 'False'; S7_SetPoint := 'False'} : R_TRIG;
      sR_TRIG_PartialBinReceived_30 {InstructionName := 'R_TRIG'; LibVersion := '1.0'; ExternalAccessible := 'False'; ExternalVisible := 'False'; ExternalWritable := 'False'; S7_SetPoint := 'False'} : R_TRIG;
      sR_TRIG_InicializeWS {InstructionName := 'R_TRIG'; LibVersion := '1.0'; ExternalAccessible := 'False'; ExternalVisible := 'False'; ExternalWritable := 'False'; S7_SetPoint := 'False'} : R_TRIG;
      sF_TRIG_StationDeactivated {InstructionName := 'F_TRIG'; LibVersion := '1.0'; ExternalAccessible := 'False'; ExternalVisible := 'False'; ExternalWritable := 'False'; S7_SetPoint := 'False'} : F_TRIG;
      sx_Counter { ExternalAccessible := 'False'; ExternalVisible := 'False'; ExternalWritable := 'False'} : Int;
      sx_StartClearing { ExternalAccessible := 'False'; ExternalVisible := 'False'; ExternalWritable := 'False'} : Bool;
      sx_Hold080 { ExternalAccessible := 'False'; ExternalVisible := 'False'; ExternalWritable := 'False'} : Bool;
      sx_ReleaseBinHoldLeft { ExternalAccessible := 'False'; ExternalVisible := 'False'; ExternalWritable := 'False'} : Bool;
      sx_ReleaseBinHoldRight { ExternalAccessible := 'False'; ExternalVisible := 'False'; ExternalWritable := 'False'} : Bool;
      sFB_TimerOnOffDelayReceiveBin { ExternalAccessible := 'False'; ExternalVisible := 'False'; ExternalWritable := 'False'; S7_SetPoint := 'False'} : "FB_TimerOnOffDelay";
      si_BinReleaseDistanceLeft { ExternalAccessible := 'False'; ExternalVisible := 'False'; ExternalWritable := 'False'} : Int;
      si_BinReleaseDistanceRight { ExternalAccessible := 'False'; ExternalVisible := 'False'; ExternalWritable := 'False'} : Int;
      sx_Hold050 { ExternalAccessible := 'False'; ExternalVisible := 'False'; ExternalWritable := 'False'} : Bool;
      sx_Hold060 { ExternalAccessible := 'False'; ExternalVisible := 'False'; ExternalWritable := 'False'} : Bool;
      sx_Hold070 { ExternalAccessible := 'False'; ExternalVisible := 'False'; ExternalWritable := 'False'} : Bool;
      sx_Hold150 { ExternalAccessible := 'False'; ExternalVisible := 'False'; ExternalWritable := 'False'} : Bool;
      sx_Hold160 { ExternalAccessible := 'False'; ExternalVisible := 'False'; ExternalWritable := 'False'} : Bool;
      sx_Hold170 { ExternalAccessible := 'False'; ExternalVisible := 'False'; ExternalWritable := 'False'} : Bool;
      sx_Hold180 { ExternalAccessible := 'False'; ExternalVisible := 'False'; ExternalWritable := 'False'} : Bool;
      sx_BinReleaseLeft { ExternalAccessible := 'False'; ExternalVisible := 'False'; ExternalWritable := 'False'} : Bool;
      sx_BinReleaseRight { ExternalAccessible := 'False'; ExternalVisible := 'False'; ExternalWritable := 'False'} : Bool;
      sFB_TimerOnOffDelay210 { ExternalAccessible := 'False'; ExternalVisible := 'False'; ExternalWritable := 'False'; S7_SetPoint := 'False'} : "FB_TimerOnOffDelay";
      sFB_TimerOnOffDelay220 { ExternalAccessible := 'False'; ExternalVisible := 'False'; ExternalWritable := 'False'; S7_SetPoint := 'False'} : "FB_TimerOnOffDelay";
      sFB_TimerOnOffDelay230 { ExternalAccessible := 'False'; ExternalVisible := 'False'; ExternalWritable := 'False'; S7_SetPoint := 'False'} : "FB_TimerOnOffDelay";
      sx_LastReleaseLeft { ExternalAccessible := 'False'; ExternalVisible := 'False'; ExternalWritable := 'False'} : Bool;
      sx_LastReleaseRight { ExternalAccessible := 'False'; ExternalVisible := 'False'; ExternalWritable := 'False'} : Bool;
      sx_Clear050 { ExternalAccessible := 'False'; ExternalVisible := 'False'; ExternalWritable := 'False'} : Bool;
      sx_Clear060 { ExternalAccessible := 'False'; ExternalVisible := 'False'; ExternalWritable := 'False'} : Bool;
      sx_Clear070 { ExternalAccessible := 'False'; ExternalVisible := 'False'; ExternalWritable := 'False'} : Bool;
      sx_Clear150 { ExternalAccessible := 'False'; ExternalVisible := 'False'; ExternalWritable := 'False'} : Bool;
      sx_Clear160 { ExternalAccessible := 'False'; ExternalVisible := 'False'; ExternalWritable := 'False'} : Bool;
      sx_Clear170 { ExternalAccessible := 'False'; ExternalVisible := 'False'; ExternalWritable := 'False'} : Bool;
   END_VAR

   VAR_TEMP
      tUDT_DummyInterface : "UDT_ConveyorInterface";   // Dummy interface structure
      tUDT_DummyVFDStatistics : "UDT_VfdStatistics";   // Dummy statistics structure
      tUDT_dummyHandshake : "UDT_ConveyorHandshake";   // Dummy handshake structure
      tUDT_FifoStatusEmpty : "UDT_FifoStatus";
      tUDT_FifoStatusPartial : "UDT_FifoStatus";
      tUDT_DummyBladeStop : "UDT_ValveInterface";
      tx_Enable : Bool;   // Enable bit
      tx_Error : Bool;
      tx_Warning : Bool;
      ts_Barcode : String;
      ti_NumberOfBinInQueue : Int;
      tx_ArraySize : Int;
   END_VAR


BEGIN
	(*
	----------------------------------------------------------------------------------------

	Version history:
	Date        | Version   | Author        | Remark
	----------------------------------------------------------------------------------------
	12/02/2023  | 4.0       | K.Pokorski    | First Release TIA 17.5
	08/06/2023  | 4.1       | S.Nieswiec    | New RAT, MCO, Displacement
	*)

	REGION Station flow control

	    REGION Timeout

	        #sFB_OperationTimeout(iudi_OnDelayTime := #iqUDT_Configuration.GlobalConfig.OperationTimeout,
	                              ix_SignalToDelay := NOT #sx_NoOperationInProgress
	                              AND #iqUDT_WorkstationCommonStatus."030".AutoON
	                              AND #iqUDT_WorkstationCommonStatus."130".AutoON
	                              AND #iqUDT_WorkstationCommonStatus."230".AutoON
	                              AND #iqUDT_WorkstationCommonStatus."040".AutoON
	                              AND #iqUDT_WorkstationCommonStatus."041".AutoON
	                              AND #iqUDT_WorkstationCommonStatus."140".AutoON
	                              AND #iqUDT_WorkstationCommonStatus."141".AutoON
	                              AND #iqUDT_WorkstationCommonStatus."240".AutoON
	                              AND #iqUDT_WorkstationCommonStatus."241".AutoON
	                              AND #iqUDT_WorkstationCommonStatus."050".AutoON
	                              AND #iqUDT_WorkstationCommonStatus."150".AutoON
	                              AND #iqUDT_WorkstationCommonStatus."250".AutoON);

	    END_REGION

	    REGION Request bin to workstation
	        // If new request from outside is received incerase counter. Counter is stored until parcel is send to proper destination. After inccreasing counter, reset request.
	        // Request 1 mean empty bin is required. Request 2 mean partialy full bin is required

	        IF #iqi_Request030 = 1 THEN

	            #si_EmptyBinRequiredCounter0X0 += 1;
	            #iqi_Request030 := 0;

	        ELSIF #iqi_Request030 = 2 THEN

	            #si_PartialyBinRequiredCounter0X0 += 1;
	            #iqi_Request030 := 0;

	        END_IF;

	        IF #iqi_Request130 = 1 THEN

	            #si_EmptyBinRequiredCounter1X0 += 1;
	            #iqi_Request130 := 0;

	        ELSIF #iqi_Request130 = 2 THEN

	            #si_PartialyBinRequiredCounter1X0 += 1;
	            #iqi_Request130 := 0;

	        END_IF;

	    END_REGION

	    REGION Send Bin form 0X0

	        // When no operation is proceed check if any operation is required. If yes then send bin with destination and start sending procedure.

	        IF #sx_NoOperationInProgress AND NOT #iqUDT_WorkstationStatus."030".PEC_EoS.PEC THEN

	            IF #iqUDT_WorkstationStatus."050".PEC_EoS.PEC AND #si_EmptyBinRequiredCounter0X0 >= 1 AND #iqUDT_Configuration.GlobalConfig.LeftStationAvailable AND #ix_StationActive THEN

	                #sx_Enable0X0In := TRUE;

	                #si_040DestinationA := 1;
	                #si_040DestinationB := 0;
	                #si_040DestinationC := 0;
	                #si_040DestinationD := 0;

	                #si_140DestinationA := 0;
	                #si_140DestinationB := 0;
	                #si_140DestinationC := 0;
	                #si_140DestinationD := 0;

	                #si_240DestinationA := 0;
	                #si_240DestinationB := 0;
	                #si_240DestinationC := 0;
	                #si_240DestinationD := 0;

	                #sx_Hold030 := FALSE;
	                #sx_Hold130 := TRUE;
	                #sx_Hold020 := TRUE;

	                #sx_NoOperationInProgress := FALSE;
	                #si_EmptyBinRequiredCounter0X0 -= 1;
	                #si_SendTo0X0 := TRUE;

	                #si_ReqestNewEmptyBin += 1;

	            ELSIF #iqUDT_WorkstationStatus."150".PEC_EoS.PEC AND #si_EmptyBinRequiredCounter1X0 >= 1 AND #iqUDT_Configuration.GlobalConfig.RightStationAvailable AND #ix_StationActive THEN

	                #sx_Enable0X0In := TRUE;

	                #si_040DestinationA := 2;
	                #si_040DestinationB := 0;
	                #si_040DestinationC := 0;
	                #si_040DestinationD := 0;

	                #si_140DestinationA := 0;
	                #si_140DestinationB := 0;
	                #si_140DestinationC := 2;
	                #si_140DestinationD := 0;

	                #si_240DestinationA := 0;
	                #si_240DestinationB := 0;
	                #si_240DestinationC := 0;
	                #si_240DestinationD := 2;

	                #sx_Hold030 := FALSE;
	                #sx_Hold130 := TRUE;
	                #sx_Hold020 := TRUE;

	                #sx_NoOperationInProgress := FALSE;
	                #si_EmptyBinRequiredCounter1X0 -= 1;
	                #si_SendTo1X0 := True;

	                #si_ReqestNewEmptyBin += 1;

	            END_IF;

	        END_IF;

	    END_REGION

	    REGION Send Bin form 1X0

	        // When no operation is proceed check if any operation is required. If yes then send bin with destination and start sending procedure.
	        IF #sx_NoOperationInProgress AND NOT #iqUDT_WorkstationStatus."130".PEC_EoS.PEC THEN

	            IF #iqUDT_WorkstationStatus."050".PEC_EoS.PEC AND #si_PartialyBinRequiredCounter0X0 >= 1 AND #iqUDT_Configuration.GlobalConfig.LeftStationAvailable AND #ix_StationActive THEN

	                #sx_Enable1X0In := TRUE;

	                #si_040DestinationA := 0;
	                #si_040DestinationB := 0;
	                #si_040DestinationC := 0;
	                #si_040DestinationD := 1;

	                #si_140DestinationA := 1;
	                #si_140DestinationB := 0;
	                #si_140DestinationC := 0;
	                #si_140DestinationD := 0;

	                #si_240DestinationA := 0;
	                #si_240DestinationB := 0;
	                #si_240DestinationC := 1;
	                #si_240DestinationD := 0;

	                #sx_Hold130 := FALSE;
	                #sx_Hold030 := TRUE;
	                #sx_Hold120 := TRUE;

	                #sx_NoOperationInProgress := FALSE;
	                #si_PartialyBinRequiredCounter0X0 -= 1;
	                #si_SendTo0X0 := TRUE;

	                #si_ReqestNewPartialBin += 1;

	            ELSIF #iqUDT_WorkstationStatus."150".PEC_EoS.PEC AND #si_PartialyBinRequiredCounter1X0 >= 1 AND #iqUDT_Configuration.GlobalConfig.RightStationAvailable AND #ix_StationActive THEN

	                #sx_Enable1X0In := TRUE;
	                #si_040DestinationA := 0;
	                #si_040DestinationB := 0;
	                #si_040DestinationC := 0;
	                #si_040DestinationD := 0;

	                #si_140DestinationA := 2;
	                #si_140DestinationB := 0;
	                #si_140DestinationC := 0;
	                #si_140DestinationD := 0;

	                #si_240DestinationA := 0;
	                #si_240DestinationB := 0;
	                #si_240DestinationC := 0;
	                #si_240DestinationD := 0;


	                #sx_Hold130 := FALSE;
	                #sx_Hold030 := TRUE;
	                #sx_Hold120 := TRUE;

	                #sx_NoOperationInProgress := FALSE;
	                #si_PartialyBinRequiredCounter1X0 -= 1;
	                #si_SendTo1X0 := TRUE;

	                #si_ReqestNewPartialBin += 1;

	            END_IF;

	        END_IF;



	    END_REGION

	    REGION Send Bin form 2X0

	        // When no operation is proceed check if any operation is required. If yes then send bin with destination and start sending procedure.

	        IF #sx_NoOperationInProgress AND NOT #iqUDT_WorkstationStatus."230".PEC_EoS.PEC AND #iqUDT_WorkstationStatus."250".PEC_EoS.PEC AND #ix_StationActive THEN


	            #sx_Enable2X0In := TRUE;


	            #si_040DestinationA := 0;
	            #si_040DestinationB := 0;
	            #si_040DestinationC := 0;
	            #si_040DestinationD := 0;

	            #si_140DestinationA := 0;
	            #si_140DestinationB := 0;
	            #si_140DestinationC := 0;
	            #si_140DestinationD := 0;

	            #si_240DestinationA := 3;
	            #si_240DestinationB := 0;
	            #si_240DestinationC := 0;
	            #si_240DestinationD := 0;


	            //  #sx_Hold130 := TRUE;
	            //   #sx_Hold030 := TRUE;
	            #sx_Hold230 := FALSE;
	            #sx_Hold220 := TRUE;


	            #sx_NoOperationInProgress := FALSE;
	            #si_SendTo2X0 := TRUE;

	        END_IF;



	    END_REGION

	    REGION Send bin to outfeed from work place
	        #sFB_TimerOnOffDelay210(iudi_OnDelayTime := 4000,
	                                ix_SignalToDelay := #iqUDT_WorkstationStatus."210".PEC_EoS.PEC);
	        #sFB_TimerOnOffDelay220(iudi_OnDelayTime := 4000,
	                                ix_SignalToDelay := #iqUDT_WorkstationStatus."220".PEC_EoS.PEC);
	        #sFB_TimerOnOffDelay230(iudi_OnDelayTime := 4000,
	                                ix_SignalToDelay := #iqUDT_WorkstationStatus."230".PEC_EoS.PEC);

	        IF NOT #sx_LastReleaseLeft
	            OR (NOT #iqx_ReleaseBin150
	            AND NOT #iqx_ReleaseBin160
	            AND NOT #iqx_ReleaseBin170)
	        THEN
	            IF (#iqx_ReleaseBin050
	                OR #iqx_ReleaseBin060
	                OR #iqx_ReleaseBin070)
	                AND NOT #sx_BinReleaseLeft
	                AND NOT #sx_BinReleaseRight
	                AND #sFB_TimerOnOffDelay210.qx_DelayedSignal
	                AND #sFB_TimerOnOffDelay220.qx_DelayedSignal
	                AND #sFB_TimerOnOffDelay230.qx_DelayedSignal
	            THEN
	                #sx_BinReleaseLeft := TRUE;
	                #sx_LastReleaseLeft := TRUE;

	                IF #iqx_ReleaseBin050 THEN
	                    #sx_Clear050 := TRUE;
	                    #iqx_ReleaseBin050 := FALSE;
	                    #tx_ArraySize := "FC_GetNrOfArrayEl"(#sa_TrackingArray_050);
	                    FILL_BLK(IN := 0,
	                             COUNT := INT_TO_ULINT(#tx_ArraySize),
	                             OUT => #sa_TrackingArray_050[0]);
	                END_IF;

	                IF #iqx_ReleaseBin060 THEN
	                    #sx_Clear060 := TRUE;
	                    #iqx_ReleaseBin060 := FALSE;
	                    #tx_ArraySize := "FC_GetNrOfArrayEl"(#sa_TrackingArray_060);
	                    FILL_BLK(IN := 0,
	                             COUNT := INT_TO_ULINT(#tx_ArraySize),
	                             OUT => #sa_TrackingArray_060[0]);
	                END_IF;

	                IF #iqx_ReleaseBin070 THEN
	                    #sx_Clear070 := TRUE;
	                    #iqx_ReleaseBin070 := FALSE;
	                    #tx_ArraySize := "FC_GetNrOfArrayEl"(#sa_TrackingArray_070);
	                    FILL_BLK(IN := 0,
	                             COUNT := INT_TO_ULINT(#tx_ArraySize),
	                             OUT => #sa_TrackingArray_070[0]);
	                END_IF;
	            END_IF;

	        END_IF;

	        IF (#iqx_ReleaseBin150
	            OR #iqx_ReleaseBin160
	            OR #iqx_ReleaseBin170)
	            AND NOT #sx_BinReleaseLeft
	            AND NOT #sx_BinReleaseRight
	            AND #sFB_TimerOnOffDelay210.qx_DelayedSignal
	            AND #sFB_TimerOnOffDelay220.qx_DelayedSignal
	            AND #sFB_TimerOnOffDelay230.qx_DelayedSignal

	        THEN
	            #sx_BinReleaseRight := TRUE;
	            #sx_LastReleaseLeft := FALSE;

	            IF #iqx_ReleaseBin150 THEN
	                #sx_Clear150 := TRUE;
	                #iqx_ReleaseBin150 := FALSE;
	                #tx_ArraySize := "FC_GetNrOfArrayEl"(#sa_TrackingArray_150);
	                FILL_BLK(IN := 0,
	                         COUNT := INT_TO_ULINT(#tx_ArraySize),
	                         OUT => #sa_TrackingArray_150[0]);
	            END_IF;

	            IF #iqx_ReleaseBin160 THEN
	                #sx_Clear160 := TRUE;
	                #iqx_ReleaseBin160 := FALSE;
	                #tx_ArraySize := "FC_GetNrOfArrayEl"(#sa_TrackingArray_160);
	                FILL_BLK(IN := 0,
	                         COUNT := INT_TO_ULINT(#tx_ArraySize),
	                         OUT => #sa_TrackingArray_160[0]);
	            END_IF;

	            IF #iqx_ReleaseBin170 THEN
	                #sx_Clear170 := TRUE;
	                #iqx_ReleaseBin170 := FALSE;
	                #tx_ArraySize := "FC_GetNrOfArrayEl"(#sa_TrackingArray_170);
	                FILL_BLK(IN := 0,
	                         COUNT := INT_TO_ULINT(#tx_ArraySize),
	                         OUT => #sa_TrackingArray_170[0]);
	            END_IF;


	        END_IF;

	        //Send from left station
	        IF #sx_BinReleaseLeft AND #iqUDT_WorkstationStatus."210".PEC_EoS.PEC
	            AND #iqUDT_WorkstationStatus."220".PEC_EoS.PEC
	            AND #iqUDT_WorkstationStatus."230".PEC_EoS.PEC
	        THEN

	            #sx_Hold080 := FALSE;
	            #sx_ReleaseBinHoldLeft := TRUE;
	            #si_BinReleaseDistanceLeft := #iqUDT_Configuration.GlobalConfig.BinReleaseDistance;
	        END_IF;
	        IF NOT #sx_BinReleaseLeft AND NOT #sx_StartClearing THEN
	            #sx_Hold080 := true;
	        END_IF;


	        IF #sx_BinReleaseLeft
	            AND (NOT #iqUDT_WorkstationStatus."210".PEC_EoS.PEC OR NOT #sx_Clear070)
	            AND (NOT #iqUDT_WorkstationStatus."220".PEC_EoS.PEC OR NOT #sx_Clear060)
	            AND (NOT #iqUDT_WorkstationStatus."230".PEC_EoS.PEC OR NOT #sx_Clear050)
	        THEN

	            #si_BinReleaseDistanceLeft -= ABS(#sUDT_Interface_080.Displacement);

	            IF #si_BinReleaseDistanceLeft <= 0 THEN

	                #sx_Hold080 := TRUE;
	                #sx_ReleaseBinHoldLeft := FALSE;
	                #sx_BinReleaseLeft := FALSE;
	                #sx_Clear050 := false;
	                #sx_Clear060 := false;
	                #sx_Clear070 := false;
	                #si_EmptyBinRequiredCounter0X0 := 2;
	                #si_PartialyBinRequiredCounter0X0 := 1;

	                IF NOT #iqUDT_WorkstationStatus."050".PEC_EoS.PEC THEN
	                    IF #sa_TrackingArray_050[#iqUDT_Configuration."050".PEC_EoS.Distance / 10 - 2] > #iqUDT_Configuration.GlobalConfig.GINRangeStart
	                        AND #sa_TrackingArray_050[#iqUDT_Configuration."050".PEC_EoS.Distance / 10 - 2] < ((#iqUDT_Configuration.GlobalConfig.GINRangeStart + #iqUDT_Configuration.GlobalConfig.GINRangeEnd) / 2) THEN
	                        IF #si_EmptyBinRequiredCounter0X0 > 0 THEN
	                            #si_EmptyBinRequiredCounter0X0 -= 1;
	                        END_IF;
	                    ELSE

	                        IF #si_PartialyBinRequiredCounter0X0 > 0 THEN
	                            #si_PartialyBinRequiredCounter0X0 -= 1;
	                        ELSE
	                            IF #si_EmptyBinRequiredCounter0X0 > 0 THEN
	                                #si_EmptyBinRequiredCounter0X0 -= 1;
	                            END_IF;


	                        END_IF;

	                    END_IF;


	                END_IF;
	                IF NOT #iqUDT_WorkstationStatus."060".PEC_EoS.PEC THEN
	                    IF #sa_TrackingArray_060[#iqUDT_Configuration."060".PEC_EoS.Distance / 10 - 2] > #iqUDT_Configuration.GlobalConfig.GINRangeStart
	                        AND #sa_TrackingArray_060[#iqUDT_Configuration."060".PEC_EoS.Distance / 10 - 2] < ((#iqUDT_Configuration.GlobalConfig.GINRangeStart + #iqUDT_Configuration.GlobalConfig.GINRangeEnd) / 2) THEN
	                        IF #si_EmptyBinRequiredCounter0X0 > 0 THEN
	                            #si_EmptyBinRequiredCounter0X0 -= 1;
	                        END_IF;
	                    ELSE

	                        IF #si_PartialyBinRequiredCounter0X0 > 0 THEN
	                            #si_PartialyBinRequiredCounter0X0 -= 1;
	                        ELSE
	                            IF #si_EmptyBinRequiredCounter0X0 > 0 THEN
	                                #si_EmptyBinRequiredCounter0X0 -= 1;
	                            END_IF;


	                        END_IF;

	                    END_IF;


	                END_IF;
	                IF NOT #iqUDT_WorkstationStatus."070".PEC_EoS.PEC THEN
	                    IF #sa_TrackingArray_070[#iqUDT_Configuration."070".PEC_EoS.Distance / 10 - 2] > #iqUDT_Configuration.GlobalConfig.GINRangeStart
	                        AND #sa_TrackingArray_070[#iqUDT_Configuration."070".PEC_EoS.Distance / 10 - 2] < ((#iqUDT_Configuration.GlobalConfig.GINRangeStart + #iqUDT_Configuration.GlobalConfig.GINRangeEnd) / 2) THEN
	                        IF #si_EmptyBinRequiredCounter0X0 > 0 THEN
	                            #si_EmptyBinRequiredCounter0X0 -= 1;
	                        END_IF;
	                    ELSE

	                        IF #si_PartialyBinRequiredCounter0X0 > 0 THEN
	                            #si_PartialyBinRequiredCounter0X0 -= 1;
	                        ELSE
	                            IF #si_EmptyBinRequiredCounter0X0 > 0 THEN
	                                #si_EmptyBinRequiredCounter0X0 -= 1;
	                            END_IF;


	                        END_IF;

	                    END_IF;


	                END_IF;
	            END_IF;

	        END_IF;


	        //Send from right station
	        IF #sx_BinReleaseRight AND #iqUDT_WorkstationStatus."210".PEC_EoS.PEC
	            AND #iqUDT_WorkstationStatus."220".PEC_EoS.PEC
	            AND #iqUDT_WorkstationStatus."230".PEC_EoS.PEC
	        THEN

	            #sx_Hold180 := FALSE;
	            #sx_ReleaseBinHoldRight := TRUE;
	            #si_BinReleaseDistanceRight := #iqUDT_Configuration.GlobalConfig.BinReleaseDistance;
	        END_IF;
	        IF NOT #sx_BinReleaseRight AND NOT #sx_StartClearing THEN
	            #sx_Hold180 := true;
	        END_IF;


	        IF #sx_BinReleaseRight
	            AND (NOT #iqUDT_WorkstationStatus."210".PEC_EoS.PEC OR NOT #sx_Clear170)
	            AND (NOT #iqUDT_WorkstationStatus."220".PEC_EoS.PEC OR NOT #sx_Clear160)
	            AND (NOT #iqUDT_WorkstationStatus."230".PEC_EoS.PEC OR NOT #sx_Clear150)
	        THEN

	            #si_BinReleaseDistanceRight -= ABS(#sUDT_Interface_180.Displacement);

	            IF #si_BinReleaseDistanceRight <= 0 THEN

	                #sx_Hold180 := TRUE;
	                #sx_ReleaseBinHoldRight := FALSE;
	                #sx_BinReleaseRight := FALSE;
	                #sx_Clear150 := false;
	                #sx_Clear160 := false;
	                #sx_Clear170 := false;
	                #si_EmptyBinRequiredCounter1X0 := 2;
	                #si_PartialyBinRequiredCounter1X0 := 1;

	                IF NOT #iqUDT_WorkstationStatus."150".PEC_EoS.PEC THEN
	                    IF #sa_TrackingArray_150[#iqUDT_Configuration."150".PEC_EoS.Distance / 10 - 2] > #iqUDT_Configuration.GlobalConfig.GINRangeStart
	                        AND #sa_TrackingArray_150[#iqUDT_Configuration."150".PEC_EoS.Distance / 10 - 2] < ((#iqUDT_Configuration.GlobalConfig.GINRangeStart + #iqUDT_Configuration.GlobalConfig.GINRangeEnd) / 2) THEN
	                        IF #si_EmptyBinRequiredCounter1X0 > 0 THEN
	                            #si_EmptyBinRequiredCounter1X0 -= 1;
	                        END_IF;
	                    ELSE

	                        IF #si_PartialyBinRequiredCounter1X0 > 0 THEN
	                            #si_PartialyBinRequiredCounter1X0 -= 1;
	                        ELSE
	                            IF #si_EmptyBinRequiredCounter1X0 > 0 THEN
	                                #si_EmptyBinRequiredCounter1X0 -= 1;
	                            END_IF;


	                        END_IF;

	                    END_IF;


	                END_IF;
	                IF NOT #iqUDT_WorkstationStatus."160".PEC_EoS.PEC THEN
	                    IF #sa_TrackingArray_160[#iqUDT_Configuration."160".PEC_EoS.Distance / 10 - 2] > #iqUDT_Configuration.GlobalConfig.GINRangeStart
	                        AND #sa_TrackingArray_160[#iqUDT_Configuration."160".PEC_EoS.Distance / 10 - 2] < ((#iqUDT_Configuration.GlobalConfig.GINRangeStart + #iqUDT_Configuration.GlobalConfig.GINRangeEnd) / 2) THEN
	                        IF #si_EmptyBinRequiredCounter1X0 > 0 THEN
	                            #si_EmptyBinRequiredCounter1X0 -= 1;
	                        END_IF;
	                    ELSE

	                        IF #si_PartialyBinRequiredCounter1X0 > 0 THEN
	                            #si_PartialyBinRequiredCounter1X0 -= 1;
	                        ELSE
	                            IF #si_EmptyBinRequiredCounter1X0 > 0 THEN
	                                #si_EmptyBinRequiredCounter1X0 -= 1;
	                            END_IF;


	                        END_IF;

	                    END_IF;


	                END_IF;
	                IF NOT #iqUDT_WorkstationStatus."170".PEC_EoS.PEC THEN
	                    IF #sa_TrackingArray_170[#iqUDT_Configuration."170".PEC_EoS.Distance / 10 - 2] > #iqUDT_Configuration.GlobalConfig.GINRangeStart
	                        AND #sa_TrackingArray_170[#iqUDT_Configuration."170".PEC_EoS.Distance / 10 - 2] < ((#iqUDT_Configuration.GlobalConfig.GINRangeStart + #iqUDT_Configuration.GlobalConfig.GINRangeEnd) / 2) THEN
	                        IF #si_EmptyBinRequiredCounter1X0 > 0 THEN
	                            #si_EmptyBinRequiredCounter1X0 -= 1;
	                        END_IF;
	                    ELSE

	                        IF #si_PartialyBinRequiredCounter1X0 > 0 THEN
	                            #si_PartialyBinRequiredCounter1X0 -= 1;
	                        ELSE
	                            IF #si_EmptyBinRequiredCounter1X0 > 0 THEN
	                                #si_EmptyBinRequiredCounter1X0 -= 1;
	                            END_IF;


	                        END_IF;

	                    END_IF;


	                END_IF;
	            END_IF;

	        END_IF;


	        //     //Send from right station
	        //     IF #sx_BinReleaseRight AND #iqUDT_WorkstationStatus."210".PEC_EoS.PEC
	        //         AND #iqUDT_WorkstationStatus."220".PEC_EoS.PEC
	        //         AND #iqUDT_WorkstationStatus."230".PEC_EoS.PEC
	        //     THEN

	        //         #sx_Hold180 := FALSE;
	        //         #sx_ReleaseBinHoldRight := TRUE;
	        //         #sx_Hold170 := TRUE;
	        //         #si_BinReleaseDistanceRight := #iUDT_Configuration.GlobalConfig.BinReleaseDistance;
	        //     END_IF;
	        //     IF NOT #sx_BinReleaseRight THEN
	        //         #sx_Hold180 := true;
	        //     END_IF;


	        //     IF #sx_BinReleaseRight
	        //         AND (NOT #iqUDT_WorkstationStatus."210".PEC_EoS.PEC
	        //         OR NOT #iqUDT_WorkstationStatus."220".PEC_EoS.PEC
	        //         OR NOT #iqUDT_WorkstationStatus."230".PEC_EoS.PEC)
	        //     THEN

	        //         #si_BinReleaseDistanceRight -= ABS(#sUDT_Interface_180.Displacement);

